REGION Network 6: Генерация импульса 10 сек.
   RUNG wire#powerrail
      { S7_Templates := "SrcType := Int" } NE_Contact(in1 := "Time_SYS_DB".Time_Now.Second, in2 := #last_10s)
      Mod(in1 := "Time_SYS_DB".Time_Now.Second, in2 := 10, out => #cnt_10s)
      wire#w1
      { S7_Templates := "SrcType := Int" } EQ_Contact(in1 := "Time_SYS_DB".Time_Now.Second, in2 := 0)
      wire#w2
      Move(in := "Time_SYS_DB".Time_Now.Second, out1 => #last_10s)
      Coil( "pulse_10s" )
   END_RUNG
   RUNG wire#w1
      { S7_Templates := "SrcType := Int" } EQ_Contact(in1 := #cnt_10s, in2 := 0)
   END_RUNG wire#w2
   // the same network as SCL:
   #_w1 := "Time_SYS_DB".Time_Now.Second <> #last_10s;
   IF #_w1 THEN #cnt_10s := "Time_SYS_DB".Time_Now.Second MOD 10; END_IF;
   #_w2 := #_w1 AND (("Time_SYS_DB".Time_Now.Second = 0) OR (#cnt_10s = 0));
   IF #_w2 THEN #last_10s := "Time_SYS_DB".Time_Now.Second; END_IF;
   "pulse_10s" := #_w2;
END_REGION

REGION Network 7: Генерация импульса 30 сек.
   RUNG wire#powerrail
      { S7_Templates := "SrcType := Int" } NE_Contact(in1 := "Time_SYS_DB".Time_Now.Second, in2 := #last_30s)
      Mod(in1 := "Time_SYS_DB".Time_Now.Second, in2 := 30, out => #cnt_30s)
      wire#w1
      { S7_Templates := "SrcType := Int" } EQ_Contact(in1 := "Time_SYS_DB".Time_Now.Second, in2 := 0)
      wire#w2
      Move(in := "Time_SYS_DB".Time_Now.Second, out1 => #last_30s)
      Coil( "pulse_30s" )
   END_RUNG
   RUNG wire#w1
      { S7_Templates := "SrcType := Int" } EQ_Contact(in1 := #cnt_30s, in2 := 0)
   END_RUNG wire#w2
   // the same network as SCL:
   #_w1 := "Time_SYS_DB".Time_Now.Second <> #last_30s;
   IF #_w1 THEN #cnt_30s := "Time_SYS_DB".Time_Now.Second MOD 30; END_IF;
   #_w2 := #_w1 AND (("Time_SYS_DB".Time_Now.Second = 0) OR (#cnt_30s = 0));
   IF #_w2 THEN #last_30s := "Time_SYS_DB".Time_Now.Second; END_IF;
   "pulse_30s" := #_w2;
END_REGION

REGION Network 8: Генерация импульса 1 мин.
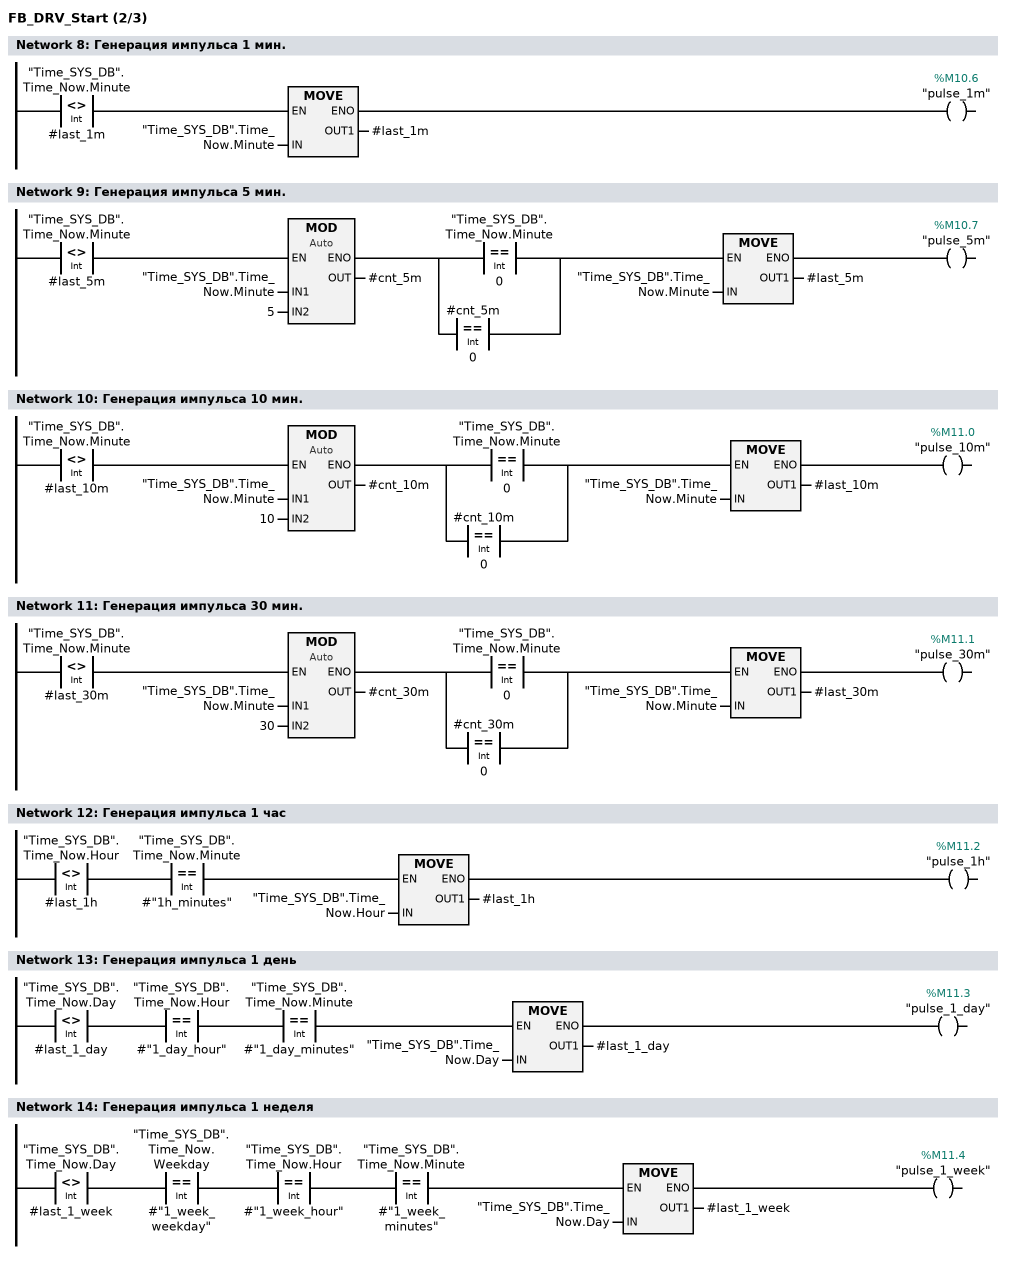
   RUNG wire#powerrail
      { S7_Templates := "SrcType := Int" } NE_Contact(in1 := "Time_SYS_DB".Time_Now.Minute, in2 := #last_1m)
      Move(in := "Time_SYS_DB".Time_Now.Minute, out1 => #last_1m)
      Coil( "pulse_1m" )
   END_RUNG
   // the same network as SCL:
   #_w1 := "Time_SYS_DB".Time_Now.Minute <> #last_1m;
   IF #_w1 THEN #last_1m := "Time_SYS_DB".Time_Now.Minute; END_IF;
   "pulse_1m" := #_w1;
END_REGION

REGION Network 9: Генерация импульса 5 мин.
   RUNG wire#powerrail
      { S7_Templates := "SrcType := Int" } NE_Contact(in1 := "Time_SYS_DB".Time_Now.Minute, in2 := #last_5m)
      Mod(in1 := "Time_SYS_DB".Time_Now.Minute, in2 := 5, out => #cnt_5m)
      wire#w1
      { S7_Templates := "SrcType := Int" } EQ_Contact(in1 := "Time_SYS_DB".Time_Now.Minute, in2 := 0)
      wire#w2
      Move(in := "Time_SYS_DB".Time_Now.Minute, out1 => #last_5m)
      Coil( "pulse_5m" )
   END_RUNG
   RUNG wire#w1
      { S7_Templates := "SrcType := Int" } EQ_Contact(in1 := #cnt_5m, in2 := 0)
   END_RUNG wire#w2
   // the same network as SCL:
   #_w1 := "Time_SYS_DB".Time_Now.Minute <> #last_5m;
   IF #_w1 THEN #cnt_5m := "Time_SYS_DB".Time_Now.Minute MOD 5; END_IF;
   #_w2 := #_w1 AND (("Time_SYS_DB".Time_Now.Minute = 0) OR (#cnt_5m = 0));
   IF #_w2 THEN #last_5m := "Time_SYS_DB".Time_Now.Minute; END_IF;
   "pulse_5m" := #_w2;
END_REGION

REGION Network 10: Генерация импульса 10 мин.
   RUNG wire#powerrail
      { S7_Templates := "SrcType := Int" } NE_Contact(in1 := "Time_SYS_DB".Time_Now.Minute, in2 := #last_10m)
      Mod(in1 := "Time_SYS_DB".Time_Now.Minute, in2 := 10, out => #cnt_10m)
      wire#w1
      { S7_Templates := "SrcType := Int" } EQ_Contact(in1 := "Time_SYS_DB".Time_Now.Minute, in2 := 0)
      wire#w2
      Move(in := "Time_SYS_DB".Time_Now.Minute, out1 => #last_10m)
      Coil( "pulse_10m" )
   END_RUNG
   RUNG wire#w1
      { S7_Templates := "SrcType := Int" } EQ_Contact(in1 := #cnt_10m, in2 := 0)
   END_RUNG wire#w2
   // the same network as SCL:
   #_w1 := "Time_SYS_DB".Time_Now.Minute <> #last_10m;
   IF #_w1 THEN #cnt_10m := "Time_SYS_DB".Time_Now.Minute MOD 10; END_IF;
   #_w2 := #_w1 AND (("Time_SYS_DB".Time_Now.Minute = 0) OR (#cnt_10m = 0));
   IF #_w2 THEN #last_10m := "Time_SYS_DB".Time_Now.Minute; END_IF;
   "pulse_10m" := #_w2;
END_REGION

REGION Network 11: Генерация импульса 30 мин.
   RUNG wire#powerrail
      { S7_Templates := "SrcType := Int" } NE_Contact(in1 := "Time_SYS_DB".Time_Now.Minute, in2 := #last_30m)
      Mod(in1 := "Time_SYS_DB".Time_Now.Minute, in2 := 30, out => #cnt_30m)
      wire#w1
      { S7_Templates := "SrcType := Int" } EQ_Contact(in1 := "Time_SYS_DB".Time_Now.Minute, in2 := 0)
      wire#w2
      Move(in := "Time_SYS_DB".Time_Now.Minute, out1 => #last_30m)
      Coil( "pulse_30m" )
   END_RUNG
   RUNG wire#w1
      { S7_Templates := "SrcType := Int" } EQ_Contact(in1 := #cnt_30m, in2 := 0)
   END_RUNG wire#w2
   // the same network as SCL:
   #_w1 := "Time_SYS_DB".Time_Now.Minute <> #last_30m;
   IF #_w1 THEN #cnt_30m := "Time_SYS_DB".Time_Now.Minute MOD 30; END_IF;
   #_w2 := #_w1 AND (("Time_SYS_DB".Time_Now.Minute = 0) OR (#cnt_30m = 0));
   IF #_w2 THEN #last_30m := "Time_SYS_DB".Time_Now.Minute; END_IF;
   "pulse_30m" := #_w2;
END_REGION

REGION Network 12: Генерация импульса 1 час
   RUNG wire#powerrail
      { S7_Templates := "SrcType := Int" } NE_Contact(in1 := "Time_SYS_DB".Time_Now.Hour, in2 := #last_1h)
      { S7_Templates := "SrcType := Int" } EQ_Contact(in1 := "Time_SYS_DB".Time_Now.Minute, in2 := #"1h_minutes")
      Move(in := "Time_SYS_DB".Time_Now.Hour, out1 => #last_1h)
      Coil( "pulse_1h" )
   END_RUNG
   // the same network as SCL:
   #_w1 := ("Time_SYS_DB".Time_Now.Hour <> #last_1h) AND ("Time_SYS_DB".Time_Now.Minute = #"1h_minutes");
   IF #_w1 THEN #last_1h := "Time_SYS_DB".Time_Now.Hour; END_IF;
   "pulse_1h" := #_w1;
END_REGION

REGION Network 13: Генерация импульса 1 день
   RUNG wire#powerrail
      { S7_Templates := "SrcType := Int" } NE_Contact(in1 := "Time_SYS_DB".Time_Now.Day, in2 := #last_1_day)
      { S7_Templates := "SrcType := Int" } EQ_Contact(in1 := "Time_SYS_DB".Time_Now.Hour, in2 := #"1_day_hour")
      { S7_Templates := "SrcType := Int" } EQ_Contact(in1 := "Time_SYS_DB".Time_Now.Minute, in2 := #"1_day_minutes")
      Move(in := "Time_SYS_DB".Time_Now.Day, out1 => #last_1_day)
      Coil( "pulse_1_day" )
   END_RUNG
   // the same network as SCL:
   #_w1 := ("Time_SYS_DB".Time_Now.Day <> #last_1_day) AND ("Time_SYS_DB".Time_Now.Hour = #"1_day_hour") AND ("Time_SYS_DB".Time_Now.Minute = #"1_day_minutes");
   IF #_w1 THEN #last_1_day := "Time_SYS_DB".Time_Now.Day; END_IF;
   "pulse_1_day" := #_w1;
END_REGION

REGION Network 14: Генерация импульса 1 неделя
   RUNG wire#powerrail
      { S7_Templates := "SrcType := Int" } NE_Contact(in1 := "Time_SYS_DB".Time_Now.Day, in2 := #last_1_week)
      { S7_Templates := "SrcType := Int" } EQ_Contact(in1 := "Time_SYS_DB".Time_Now.Weekday, in2 := #"1_week_weekday")
      { S7_Templates := "SrcType := Int" } EQ_Contact(in1 := "Time_SYS_DB".Time_Now.Hour, in2 := #"1_week_hour")
      { S7_Templates := "SrcType := Int" } EQ_Contact(in1 := "Time_SYS_DB".Time_Now.Minute, in2 := #"1_week_minutes")
      Move(in := "Time_SYS_DB".Time_Now.Day, out1 => #last_1_week)
      Coil( "pulse_1_week" )
   END_RUNG
   // the same network as SCL:
   #_w1 := ("Time_SYS_DB".Time_Now.Day <> #last_1_week) AND ("Time_SYS_DB".Time_Now.Weekday = #"1_week_weekday") AND ("Time_SYS_DB".Time_Now.Hour = #"1_week_hour") AND ("Time_SYS_DB".Time_Now.Minute = #"1_week_minutes");
   IF #_w1 THEN #last_1_week := "Time_SYS_DB".Time_Now.Day; END_IF;
   "pulse_1_week" := #_w1;
END_REGION

REGION Network 15: Генерация импульса 1 месяц
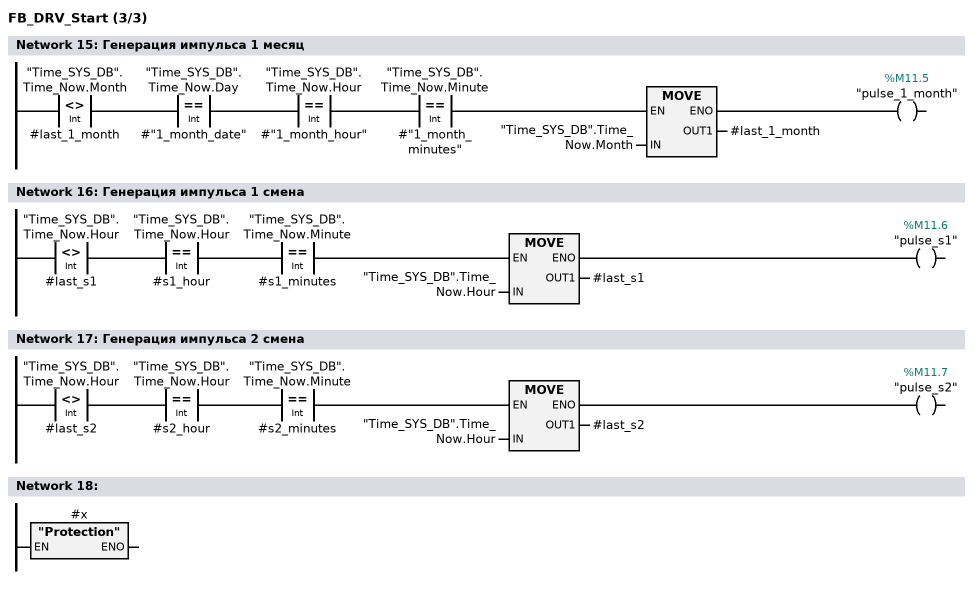
   RUNG wire#powerrail
      { S7_Templates := "SrcType := Int" } NE_Contact(in1 := "Time_SYS_DB".Time_Now.Month, in2 := #last_1_month)
      { S7_Templates := "SrcType := Int" } EQ_Contact(in1 := "Time_SYS_DB".Time_Now.Day, in2 := #"1_month_date")
      { S7_Templates := "SrcType := Int" } EQ_Contact(in1 := "Time_SYS_DB".Time_Now.Hour, in2 := #"1_month_hour")
      { S7_Templates := "SrcType := Int" } EQ_Contact(in1 := "Time_SYS_DB".Time_Now.Minute, in2 := #"1_month_minutes")
      Move(in := "Time_SYS_DB".Time_Now.Month, out1 => #last_1_month)
      Coil( "pulse_1_month" )
   END_RUNG
   // the same network as SCL:
   #_w1 := ("Time_SYS_DB".Time_Now.Month <> #last_1_month) AND ("Time_SYS_DB".Time_Now.Day = #"1_month_date") AND ("Time_SYS_DB".Time_Now.Hour = #"1_month_hour") AND ("Time_SYS_DB".Time_Now.Minute = #"1_month_minutes");
   IF #_w1 THEN #last_1_month := "Time_SYS_DB".Time_Now.Month; END_IF;
   "pulse_1_month" := #_w1;
END_REGION

REGION Network 16: Генерация импульса 1 смена
   RUNG wire#powerrail
      { S7_Templates := "SrcType := Int" } NE_Contact(in1 := "Time_SYS_DB".Time_Now.Hour, in2 := #last_s1)
      { S7_Templates := "SrcType := Int" } EQ_Contact(in1 := "Time_SYS_DB".Time_Now.Hour, in2 := #s1_hour)
      { S7_Templates := "SrcType := Int" } EQ_Contact(in1 := "Time_SYS_DB".Time_Now.Minute, in2 := #s1_minutes)
      Move(in := "Time_SYS_DB".Time_Now.Hour, out1 => #last_s1)
      Coil( "pulse_s1" )
   END_RUNG
   // the same network as SCL:
   #_w1 := ("Time_SYS_DB".Time_Now.Hour <> #last_s1) AND ("Time_SYS_DB".Time_Now.Hour = #s1_hour) AND ("Time_SYS_DB".Time_Now.Minute = #s1_minutes);
   IF #_w1 THEN #last_s1 := "Time_SYS_DB".Time_Now.Hour; END_IF;
   "pulse_s1" := #_w1;
END_REGION

REGION Network 17: Генерация импульса 2 смена
   RUNG wire#powerrail
      { S7_Templates := "SrcType := Int" } NE_Contact(in1 := "Time_SYS_DB".Time_Now.Hour, in2 := #last_s2)
      { S7_Templates := "SrcType := Int" } EQ_Contact(in1 := "Time_SYS_DB".Time_Now.Hour, in2 := #s2_hour)
      { S7_Templates := "SrcType := Int" } EQ_Contact(in1 := "Time_SYS_DB".Time_Now.Minute, in2 := #s2_minutes)
      Move(in := "Time_SYS_DB".Time_Now.Hour, out1 => #last_s2)
      Coil( "pulse_s2" )
   END_RUNG
   // the same network as SCL:
   #_w1 := ("Time_SYS_DB".Time_Now.Hour <> #last_s2) AND ("Time_SYS_DB".Time_Now.Hour = #s2_hour) AND ("Time_SYS_DB".Time_Now.Minute = #s2_minutes);
   IF #_w1 THEN #last_s2 := "Time_SYS_DB".Time_Now.Hour; END_IF;
   "pulse_s2" := #_w1;
END_REGION

REGION Network 18
   RUNG wire#powerrail
      #x()
   END_RUNG
   // the same network as SCL:
   #x();   // "Protection"
END_REGION
END_FUNCTION_BLOCK

FUNCTION_BLOCK "Time_SYS"   // FB95, LAD
{ S7_Optimized_Access := 'FALSE' }
VERSION : 0.1
// stored: AutoNumber false, IsIECCheckEnabled false, SetENOAutomatically false, UDAEnableTagReadback false
   VAR DB_SPECIFIC
      Set_Time : Bool;   // Заданное время
      Time_Now : Struct   // Текущее время
         Year : Int;   // год
         Month : Int;   // месяц
         Day : Int;   // день месяца
         Weekday : Int;   // день недели (1 - воскресенье)
         Hour : Int;   // часы
         Minute : Int;   // минуты
         Second : Int;   // секунды
      END_STRUCT;
      Time_SP : Struct   // Текущее время
         Year : Int;   // год
         Month : Int;   // месяц
         Day : Int;   // день месяца
         Weekday : Int;   // день недели (1 - воскресенье)
         Hour : Int;   // часы
         Minute : Int;   // минуты
         Second : Int;   // секунды
      END_STRUCT;
      TimeZone { S7_SetPoint := 'True'} : TimeTransformationRule;   // Часовой пояс
      RD_SYS_Status : Int;   // Статус чтения времени
      WR_SYS_Status : Int;   // Статус записи времени
      RD_Time : DTL;   // Прочитанное сист. время
      SP_Time : DTL;   // Новое сист. время
   END_VAR
   VAR
      SET_TIMEZONE { S7_SetPoint := 'True'} : SET_TIMEZONE;   // Запись часового пояса
   END_VAR
   VAR DB_SPECIFIC
      Time_DTL : DTL;
   END_VAR
   // TimeZone.Bias := 180;   // Часовой пояс по GMT (смещение в минутах)
   // TimeZone.DaylightBias := 60;
   // TimeZone.DaylightStartMonth := 3;
   // TimeZone.DaylightStartWeek := 5;
   // TimeZone.DaylightStartWeekday := 7;
   // TimeZone.DaylightStartHour := 2;
   // TimeZone.DaylightStartMinute := 0;
   // TimeZone.StandardStartMonth := 10;
   // TimeZone.StandardStartWeek := 5;
   // TimeZone.StandardStartWeekday := 1;
   // TimeZone.StandardStartHour := 3;
   // TimeZone.StandardStartMinute := 0;
   // TimeZone.TimeZoneName := 'GMT+3';
   VAR_TEMP   // added for the SCL form of the ladder/FBD networks
      _w1 : Bool;
   END_VAR
BEGIN

REGION Network 1: Чтение системного времени
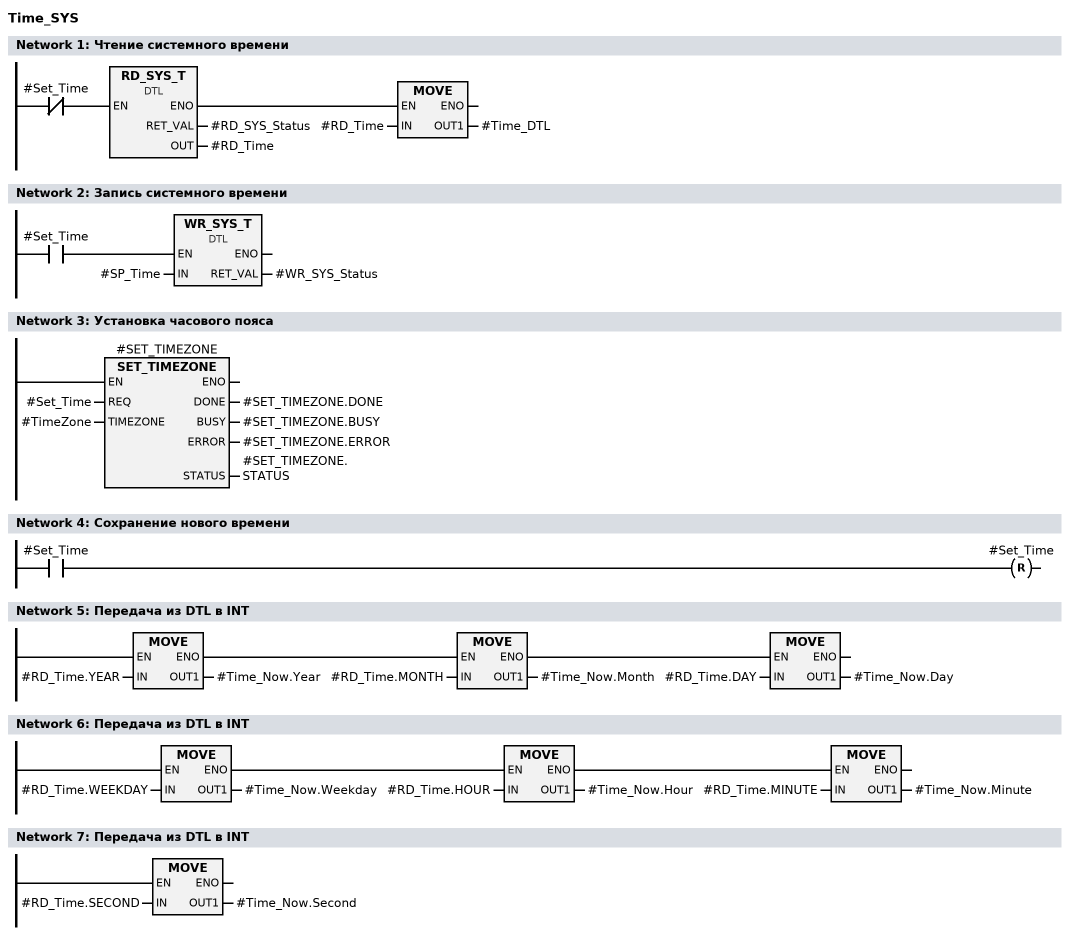
   RUNG wire#powerrail
      I_Contact( #Set_Time )
      { S7_Templates := "date_type := DTL" } RD_SYS_T(RET_VAL => #RD_SYS_Status, OUT => #RD_Time)
      Move(in := #RD_Time, out1 => #Time_DTL)
   END_RUNG
   // the same network as SCL:
   #RD_SYS_Status := RD_SYS_T(EN := NOT #Set_Time, OUT => #RD_Time, ENO => #_w1);
   IF #_w1 THEN #Time_DTL := #RD_Time; END_IF;
END_REGION

REGION Network 2: Запись системного времени
   RUNG wire#powerrail
      Contact( #Set_Time )
      { S7_Templates := "date_type := DTL" } WR_SYS_T(IN := #SP_Time, RET_VAL => #WR_SYS_Status)
   END_RUNG
   // the same network as SCL:
   IF #Set_Time THEN #WR_SYS_Status := WR_SYS_T(IN := #SP_Time); END_IF;
END_REGION

REGION Network 3: Установка часового пояса
   RUNG wire#powerrail
      #SET_TIMEZONE.SET_TIMEZONE(REQ := #Set_Time, TimeZone := #TimeZone, DONE => #SET_TIMEZONE.DONE, BUSY => #SET_TIMEZONE.BUSY, ERROR => #SET_TIMEZONE.ERROR, STATUS => #SET_TIMEZONE.STATUS)
   END_RUNG
   // the same network as SCL:
   #SET_TIMEZONE(REQ := #Set_Time,   // SET_TIMEZONE
                 TimeZone := #TimeZone,
                 DONE => #SET_TIMEZONE.DONE,
                 BUSY => #SET_TIMEZONE.BUSY,
                 ERROR => #SET_TIMEZONE.ERROR,
                 STATUS => #SET_TIMEZONE.STATUS);
END_REGION

REGION Network 4: Сохранение нового времени
   RUNG wire#powerrail
      Contact( #Set_Time )
      R_Coil( #Set_Time )
   END_RUNG
   // the same network as SCL:
   IF #Set_Time THEN #Set_Time := FALSE; END_IF;
END_REGION

REGION Network 5: Передача из DTL в INT
   RUNG wire#powerrail
      Move(in := #RD_Time.YEAR, out1 => #Time_Now.Year)
      Move(in := #RD_Time.MONTH, out1 => #Time_Now.Month)
      Move(in := #RD_Time.DAY, out1 => #Time_Now.Day)
   END_RUNG
   // the same network as SCL:
   #Time_Now.Year := #RD_Time.YEAR;
   #Time_Now.Month := #RD_Time.MONTH;
   #Time_Now.Day := #RD_Time.DAY;
END_REGION

REGION Network 6: Передача из DTL в INT
   RUNG wire#powerrail
      Move(in := #RD_Time.WEEKDAY, out1 => #Time_Now.Weekday)
      Move(in := #RD_Time.HOUR, out1 => #Time_Now.Hour)
      Move(in := #RD_Time.MINUTE, out1 => #Time_Now.Minute)
   END_RUNG
   // the same network as SCL:
   #Time_Now.Weekday := #RD_Time.WEEKDAY;
   #Time_Now.Hour := #RD_Time.HOUR;
   #Time_Now.Minute := #RD_Time.MINUTE;
END_REGION

REGION Network 7: Передача из DTL в INT
   RUNG wire#powerrail
      Move(in := #RD_Time.SECOND, out1 => #Time_Now.Second)
   END_RUNG
   // the same network as SCL:
   #Time_Now.Second := #RD_Time.SECOND;
END_REGION
END_FUNCTION_BLOCK

FUNCTION_BLOCK "Time_D"   // FB94, LAD
{ S7_Optimized_Access := 'FALSE' }
VERSION : 0.1
// stored: AutoNumber false, IsIECCheckEnabled false, SetENOAutomatically false, UDAEnableTagReadback false
   VAR DB_SPECIFIC
      SP_D { S7_SetPoint := 'True'} : DInt := 4;   // Уставка дней - от 0 до 999
      SP_H { S7_SetPoint := 'True'} : DInt;   // Уставка часов - от 0 до 23
      SP_M { S7_SetPoint := 'True'} : DInt;   // Уставка минут - от 0 до 59
      SP_S { S7_SetPoint := 'True'} : DInt;   // Уставка секунд - от 0 до 59
      Now_D : DInt;   // Прошло дней от начала отсчёта
      Now_H : DInt;   // Прошло часов от начала отсчёта
      Now_M : DInt;   // Прошло минут от начала отсчёта
      Now_S : DInt;   // Прошло секунд от начала отсчёта
      Rev_D : DInt;   // Осталось дней до уставки
      Rev_H : DInt;   // Осталось часов до уставки
      Rev_M : DInt;   // Осталось минут до уставки
      Rev_S : DInt;   // Осталось секунд до уставки
      Progress : Real;   // Прогресс выполнения
      Start : Bool;   // Запуск
      "Exit" : Bool;   // Счёт завершён
      Pause : Bool;   // Пауза
      Reset : Bool;   // Сброс таймера
   END_VAR
   VAR_TEMP
      Full_SP_S : DInt;
      Full_Now_S : DInt;
      Full_Delta_S : DInt;
      x1 : DInt;
      x2 : DInt;
   END_VAR
   VAR_TEMP   // added for the SCL form of the ladder/FBD networks
      _w1 : Bool;
      _w2 : Bool;
      _w3 : Bool;
   END_VAR
BEGIN

REGION Network 1: Подсчёт времени
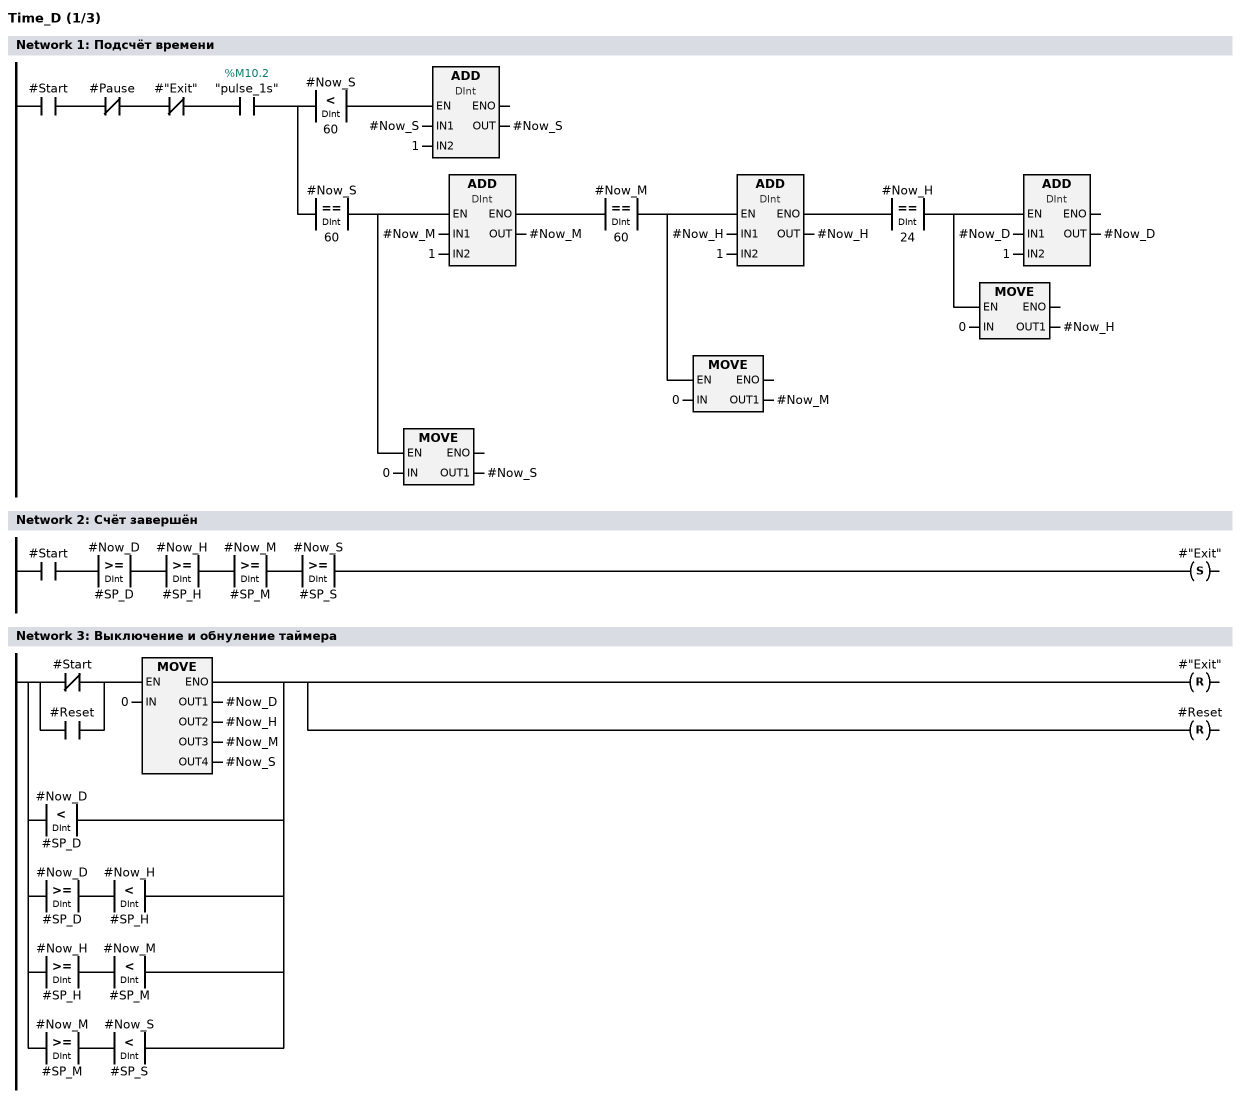
   RUNG wire#powerrail
      Contact( #Start )
      I_Contact( #Pause )
      I_Contact( #"Exit" )
      Contact( "pulse_1s" )
      wire#w1
      { S7_Templates := "SrcType := DInt" } LT_Contact(in1 := #Now_S, in2 := 60)
      { S7_Templates := "SrcType := DInt"; S7_GenerateENO := "TRUE" } Add(in1 := #Now_S, in2 := 1, out => #Now_S)
   END_RUNG
   RUNG wire#w1
      { S7_Templates := "SrcType := DInt" } EQ_Contact(in1 := #Now_S, in2 := 60)
      wire#w2
      { S7_Templates := "SrcType := DInt"; S7_GenerateENO := "TRUE" } Add(in1 := #Now_M, in2 := 1, out => #Now_M)
      { S7_Templates := "SrcType := DInt" } EQ_Contact(in1 := #Now_M, in2 := 60)
      wire#w3
      { S7_Templates := "SrcType := DInt"; S7_GenerateENO := "TRUE" } Add(in1 := #Now_H, in2 := 1, out => #Now_H)
      { S7_Templates := "SrcType := DInt" } EQ_Contact(in1 := #Now_H, in2 := 24)
      wire#w4
      { S7_Templates := "SrcType := DInt"; S7_GenerateENO := "TRUE" } Add(in1 := #Now_D, in2 := 1, out => #Now_D)
   END_RUNG
   RUNG wire#w4
      { S7_GenerateENO := "TRUE" } Move(in := 0, out1 => #Now_H)
   END_RUNG
   RUNG wire#w3
      { S7_GenerateENO := "TRUE" } Move(in := 0, out1 => #Now_M)
   END_RUNG
   RUNG wire#w2
      { S7_GenerateENO := "TRUE" } Move(in := 0, out1 => #Now_S)
   END_RUNG
   // the same network as SCL:
   // ENO of a box is taken as its EN; it also drops when the box reports an error
   #_w1 := #Start AND NOT #Pause AND NOT #"Exit" AND "pulse_1s";
   IF #_w1 AND (#Now_S < 60) THEN #Now_S := #Now_S + 1; END_IF;
   #_w2 := #_w1 AND (#Now_S = 60);
   IF #_w2 THEN #Now_M := #Now_M + 1; END_IF;
   #_w3 := #_w2 AND (#Now_M = 60);
   IF #_w3 THEN #Now_H := #Now_H + 1; END_IF;
   IF #_w3 AND (#Now_H = 24) THEN
       #Now_D := #Now_D + 1;
       #Now_H := 0;
   END_IF;
   IF #_w3 THEN #Now_M := 0; END_IF;
   IF #_w2 THEN #Now_S := 0; END_IF;
END_REGION

REGION Network 2: Счёт завершён
   RUNG wire#powerrail
      Contact( #Start )
      { S7_Templates := "SrcType := DInt" } GE_Contact(in1 := #Now_D, in2 := #SP_D)
      { S7_Templates := "SrcType := DInt" } GE_Contact(in1 := #Now_H, in2 := #SP_H)
      { S7_Templates := "SrcType := DInt" } GE_Contact(in1 := #Now_M, in2 := #SP_M)
      { S7_Templates := "SrcType := DInt" } GE_Contact(in1 := #Now_S, in2 := #SP_S)
      S_Coil( #"Exit" )
   END_RUNG
   // the same network as SCL:
   IF #Start AND (#Now_D >= #SP_D) AND (#Now_H >= #SP_H) AND (#Now_M >= #SP_M) AND (#Now_S >= #SP_S) THEN
       #"Exit" := TRUE;
   END_IF;
END_REGION

REGION Network 3: Выключение и обнуление таймера
   RUNG wire#powerrail
      I_Contact( #Start )
      wire#w1
      { S7_GenerateENO := "TRUE" } Move(in := 0, out1 => #Now_D, out2 => #Now_H, out3 => #Now_M, out4 => #Now_S)
      wire#w2
      R_Coil( #"Exit" )
   END_RUNG
   RUNG wire#powerrail
      Contact( #Reset )
   END_RUNG wire#w1
   RUNG wire#powerrail
      { S7_Templates := "SrcType := DInt" } LT_Contact(in1 := #Now_D, in2 := #SP_D)
   END_RUNG wire#w2
   RUNG wire#powerrail
      { S7_Templates := "SrcType := DInt" } GE_Contact(in1 := #Now_D, in2 := #SP_D)
      { S7_Templates := "SrcType := DInt" } LT_Contact(in1 := #Now_H, in2 := #SP_H)
   END_RUNG wire#w2
   RUNG wire#powerrail
      { S7_Templates := "SrcType := DInt" } GE_Contact(in1 := #Now_H, in2 := #SP_H)
      { S7_Templates := "SrcType := DInt" } LT_Contact(in1 := #Now_M, in2 := #SP_M)
   END_RUNG wire#w2
   RUNG wire#powerrail
      { S7_Templates := "SrcType := DInt" } GE_Contact(in1 := #Now_M, in2 := #SP_M)
      { S7_Templates := "SrcType := DInt" } LT_Contact(in1 := #Now_S, in2 := #SP_S)
   END_RUNG wire#w2
   RUNG wire#w2
      R_Coil( #Reset )
   END_RUNG
   // the same network as SCL:
   // ENO of a box is taken as its EN; it also drops when the box reports an error
   #_w1 := NOT #Start OR #Reset;
   IF #_w1 THEN
       #Now_D := 0;
       #Now_H := 0;
       #Now_M := 0;
       #Now_S := 0;
   END_IF;
   IF #_w1 OR (#Now_D < #SP_D) OR ((#Now_D >= #SP_D) AND (#Now_H < #SP_H)) OR ((#Now_H >= #SP_H) AND (#Now_M < #SP_M)) OR ((#Now_M >= #SP_M) AND (#Now_S < #SP_S)) THEN
       #"Exit" := FALSE;
       #Reset := FALSE;
   END_IF;
END_REGION

REGION Network 4: Поправка переполнения времени
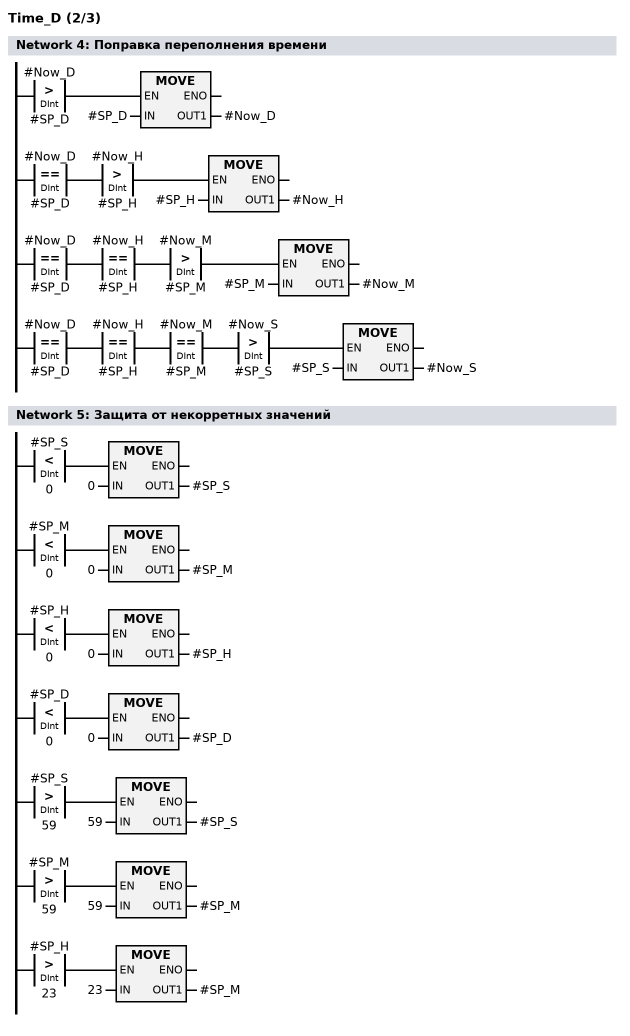
   RUNG wire#powerrail
      { S7_Templates := "SrcType := DInt" } GT_Contact(in1 := #Now_D, in2 := #SP_D)
      { S7_GenerateENO := "TRUE" } Move(in := #SP_D, out1 => #Now_D)
   END_RUNG
   RUNG wire#powerrail
      { S7_Templates := "SrcType := DInt" } EQ_Contact(in1 := #Now_D, in2 := #SP_D)
      { S7_Templates := "SrcType := DInt" } GT_Contact(in1 := #Now_H, in2 := #SP_H)
      { S7_GenerateENO := "TRUE" } Move(in := #SP_H, out1 => #Now_H)
   END_RUNG
   RUNG wire#powerrail
      { S7_Templates := "SrcType := DInt" } EQ_Contact(in1 := #Now_D, in2 := #SP_D)
      { S7_Templates := "SrcType := DInt" } EQ_Contact(in1 := #Now_H, in2 := #SP_H)
      { S7_Templates := "SrcType := DInt" } GT_Contact(in1 := #Now_M, in2 := #SP_M)
      { S7_GenerateENO := "TRUE" } Move(in := #SP_M, out1 => #Now_M)
   END_RUNG
   RUNG wire#powerrail
      { S7_Templates := "SrcType := DInt" } EQ_Contact(in1 := #Now_D, in2 := #SP_D)
      { S7_Templates := "SrcType := DInt" } EQ_Contact(in1 := #Now_H, in2 := #SP_H)
      { S7_Templates := "SrcType := DInt" } EQ_Contact(in1 := #Now_M, in2 := #SP_M)
      { S7_Templates := "SrcType := DInt" } GT_Contact(in1 := #Now_S, in2 := #SP_S)
      { S7_GenerateENO := "TRUE" } Move(in := #SP_S, out1 => #Now_S)
   END_RUNG
   // the same network as SCL:
   IF #Now_D > #SP_D THEN #Now_D := #SP_D; END_IF;
   IF (#Now_D = #SP_D) AND (#Now_H > #SP_H) THEN #Now_H := #SP_H; END_IF;
   IF (#Now_D = #SP_D) AND (#Now_H = #SP_H) AND (#Now_M > #SP_M) THEN #Now_M := #SP_M; END_IF;
   IF (#Now_D = #SP_D) AND (#Now_H = #SP_H) AND (#Now_M = #SP_M) AND (#Now_S > #SP_S) THEN
       #Now_S := #SP_S;
   END_IF;
END_REGION

REGION Network 5: Защита от некорретных значений
   RUNG wire#powerrail
      { S7_Templates := "SrcType := DInt" } LT_Contact(in1 := #SP_S, in2 := 0)
      { S7_GenerateENO := "TRUE" } Move(in := 0, out1 => #SP_S)
   END_RUNG
   RUNG wire#powerrail
      { S7_Templates := "SrcType := DInt" } LT_Contact(in1 := #SP_M, in2 := 0)
      { S7_GenerateENO := "TRUE" } Move(in := 0, out1 => #SP_M)
   END_RUNG
   RUNG wire#powerrail
      { S7_Templates := "SrcType := DInt" } LT_Contact(in1 := #SP_H, in2 := 0)
      { S7_GenerateENO := "TRUE" } Move(in := 0, out1 => #SP_H)
   END_RUNG
   RUNG wire#powerrail
      { S7_Templates := "SrcType := DInt" } LT_Contact(in1 := #SP_D, in2 := 0)
      { S7_GenerateENO := "TRUE" } Move(in := 0, out1 => #SP_D)
   END_RUNG
   RUNG wire#powerrail
      { S7_Templates := "SrcType := DInt" } GT_Contact(in1 := #SP_S, in2 := 59)
      { S7_GenerateENO := "TRUE" } Move(in := 59, out1 => #SP_S)
   END_RUNG
   RUNG wire#powerrail
      { S7_Templates := "SrcType := DInt" } GT_Contact(in1 := #SP_M, in2 := 59)
      { S7_GenerateENO := "TRUE" } Move(in := 59, out1 => #SP_M)
   END_RUNG
   RUNG wire#powerrail
      { S7_Templates := "SrcType := DInt" } GT_Contact(in1 := #SP_H, in2 := 23)
      { S7_GenerateENO := "TRUE" } Move(in := 23, out1 => #SP_M)
   END_RUNG
   // the same network as SCL:
   IF #SP_S < 0 THEN #SP_S := 0; END_IF;
   IF #SP_M < 0 THEN #SP_M := 0; END_IF;
   IF #SP_H < 0 THEN #SP_H := 0; END_IF;
   IF #SP_D < 0 THEN #SP_D := 0; END_IF;
   IF #SP_S > 59 THEN #SP_S := 59; END_IF;
   IF #SP_M > 59 THEN #SP_M := 59; END_IF;
   IF #SP_H > 23 THEN #SP_M := 23; END_IF;
END_REGION

REGION Network 6: Обратный отсчёт
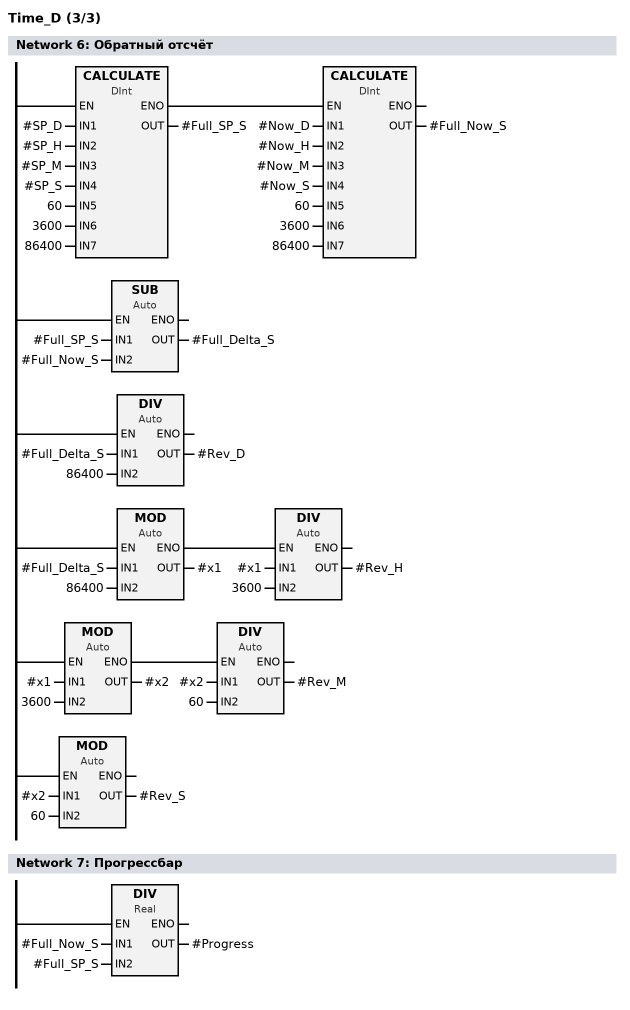
   RUNG wire#powerrail
      { S7_Templates := "SrcType := DInt"; S7_Expression := "(IN1*IN7)+(IN2*IN6)+(IN3*IN5)+IN4" } Calculate(in1 := #SP_D, in2 := #SP_H, in3 := #SP_M, in4 := #SP_S, in5 := 60, in6 := 3600, in7 := 86400, out => #Full_SP_S)
      { S7_Templates := "SrcType := DInt"; S7_Expression := "(IN1*IN7)+(IN2*IN6)+(IN3*IN5)+IN4" } Calculate(in1 := #Now_D, in2 := #Now_H, in3 := #Now_M, in4 := #Now_S, in5 := 60, in6 := 3600, in7 := 86400, out => #Full_Now_S)
   END_RUNG
   RUNG wire#powerrail
      Sub(in1 := #Full_SP_S, in2 := #Full_Now_S, out => #Full_Delta_S)
   END_RUNG
   RUNG wire#powerrail
      Div(in1 := #Full_Delta_S, in2 := 86400, out => #Rev_D)
   END_RUNG
   RUNG wire#powerrail
      Mod(in1 := #Full_Delta_S, in2 := 86400, out => #x1)
      Div(in1 := #x1, in2 := 3600, out => #Rev_H)
   END_RUNG
   RUNG wire#powerrail
      Mod(in1 := #x1, in2 := 3600, out => #x2)
      Div(in1 := #x2, in2 := 60, out => #Rev_M)
   END_RUNG
   RUNG wire#powerrail
      Mod(in1 := #x2, in2 := 60, out => #Rev_S)
   END_RUNG
   // the same network as SCL:
   #Full_SP_S := (#SP_D*86400)+(#SP_H*3600)+(#SP_M*60)+#SP_S;
   #Full_Now_S := (#Now_D*86400)+(#Now_H*3600)+(#Now_M*60)+#Now_S;
   #Full_Delta_S := #Full_SP_S - #Full_Now_S;
   #Rev_D := #Full_Delta_S / 86400;
   #x1 := #Full_Delta_S MOD 86400;
   #Rev_H := #x1 / 3600;
   #x2 := #x1 MOD 3600;
   #Rev_M := #x2 / 60;
   #Rev_S := #x2 MOD 60;
END_REGION

REGION Network 7: Прогрессбар
   RUNG wire#powerrail
      { S7_Templates := "SrcType := Real" } Div(in1 := #Full_Now_S, in2 := #Full_SP_S, out => #Progress)
   END_RUNG
   // the same network as SCL:
   #Progress := #Full_Now_S / #Full_SP_S;
END_REGION
END_FUNCTION_BLOCK

FUNCTION_BLOCK "DIx_1"   // FB200, LAD
{ S7_Optimized_Access := 'FALSE' }
VERSION : 0.1
// Input - входной сигнал контроллера
// pulse - частота фильтрации дребезга
// Signal - обработанный и отфильтрованный сигнал, используемый в дальнейшем
// stored: AutoNumber false, IsIECCheckEnabled false, SetENOAutomatically false, UDAEnableTagReadback false
   VAR
      AllBlock { S7_SetPoint := 'True'} : "DI_ex";   // Аварийный останов / 2.4 разрешение на работу
      EZ_1_FB_AHLS { S7_SetPoint := 'True'} : "DI_ex";   // Электролизер 1 (Переполнение поддона) / 2.3 Нижний уровень
      Gas_Chanel_1_1 { S7_SetPoint := 'True'} : "DI_ex";   // Загазованность канал 1 (Порог 1) / Ротаметр 1
      Gas_Chanel_1_2 { S7_SetPoint := 'True'} : "DI_ex";   // Загазованность канал 1 (Порог 2) / Ротаметр 2
      Gas_Chanel_2_1 { S7_SetPoint := 'True'} : "DI_ex";   // Загазованность канал 2 (Порог 1) / Ротаметр 3
      Gas_Chanel_2_2 { S7_SetPoint := 'True'} : "DI_ex";   // Загазованность канал 2 (Порог 2) / Датчик переливва
      ALS_1 { S7_SetPoint := 'True'} : "DI_ex";   // Аварийный уровень 1 / Датчик переливва
      KC_1 { S7_SetPoint := 'True'} : "DI_ex";   // Блок клапанов (Сигнал 1)
      KC_2 { S7_SetPoint := 'True'} : "DI_ex";   // Блок клапанов (Сигнал 2)
      signal_10 { S7_SetPoint := 'True'} : "DI_ex";
      signal_11 { S7_SetPoint := 'True'} : "DI_ex";
      signal_12 { S7_SetPoint := 'True'} : "DI_ex";
      signal_13 { S7_SetPoint := 'True'} : "DI_ex";
   END_VAR
   VAR DB_SPECIFIC
      Time_DTL { S7_SetPoint := 'True'} : DTL;
   END_VAR
   // AllBlock.ADDR_Byte := 1;
   // AllBlock.ADDR_Bit := 5;
   // EZ_1_FB_AHLS.ADDR_Byte := 0;
   // EZ_1_FB_AHLS.ADDR_Bit := 2;
   // Gas_Chanel_1_1.ADDR_Bit := 7;
   // Gas_Chanel_1_2.ADDR_Byte := 1;
   // Gas_Chanel_1_2.ADDR_Bit := 0;
   // Gas_Chanel_2_1.ADDR_Byte := 1;
   // Gas_Chanel_2_1.ADDR_Bit := 1;
   // Gas_Chanel_2_2.ADDR_Byte := 1;
   // Gas_Chanel_2_2.ADDR_Bit := 2;
   // ALS_1.ADDR_Byte := 2;
   // ALS_1.ADDR_Bit := 0;
   // KC_1.ADDR_Byte := 1;
   // KC_1.ADDR_Bit := 3;
   // KC_2.ADDR_Byte := 1;
   // KC_2.ADDR_Bit := 4;
   VAR_TEMP   // added for the SCL form of the ladder/FBD networks
      _w1 : Bool;
      _w2 : Bool;
   END_VAR
BEGIN

REGION Network 1: AllBlock
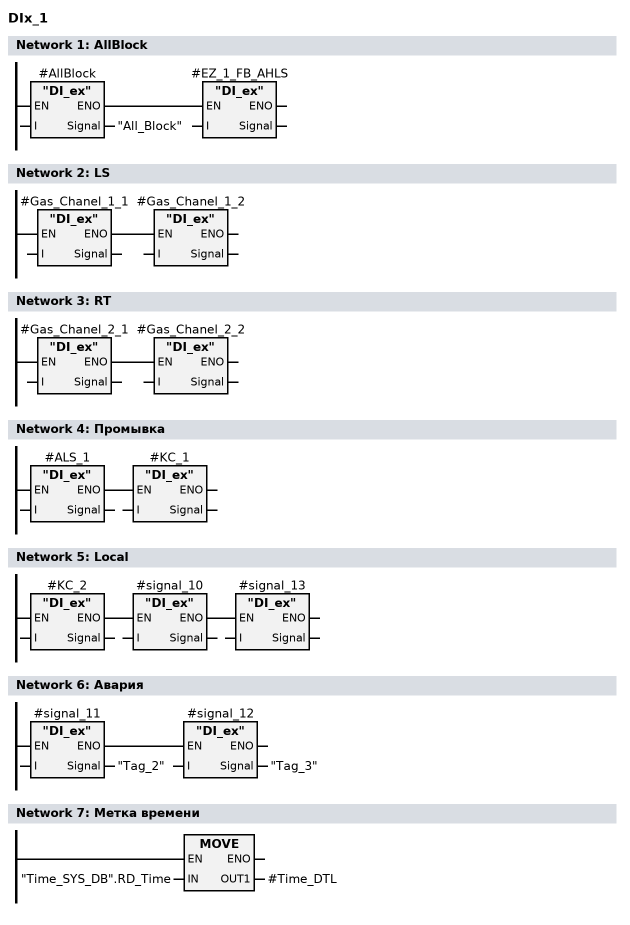
   RUNG wire#powerrail
      #AllBlock(I :=, Signal => "All_Block")
      #EZ_1_FB_AHLS(I :=, Signal =>)
   END_RUNG
   // the same network as SCL:
   #AllBlock(Signal => "All_Block", ENO => #_w1);   // "DI_ex"
   IF #_w1 THEN
       #EZ_1_FB_AHLS();   // "DI_ex"
   END_IF;
END_REGION

REGION Network 2: LS
   RUNG wire#powerrail
      #Gas_Chanel_1_1(I :=, Signal =>)
      #Gas_Chanel_1_2(I :=, Signal =>)
   END_RUNG
   // the same network as SCL:
   #Gas_Chanel_1_1(ENO => #_w1);   // "DI_ex"
   IF #_w1 THEN
       #Gas_Chanel_1_2();   // "DI_ex"
   END_IF;
END_REGION

REGION Network 3: RT
   RUNG wire#powerrail
      #Gas_Chanel_2_1(I :=, Signal =>)
      #Gas_Chanel_2_2(I :=, Signal =>)
   END_RUNG
   // the same network as SCL:
   #Gas_Chanel_2_1(ENO => #_w1);   // "DI_ex"
   IF #_w1 THEN
       #Gas_Chanel_2_2();   // "DI_ex"
   END_IF;
END_REGION

REGION Network 4: Промывка
   RUNG wire#powerrail
      #ALS_1(I :=, Signal =>)
      #KC_1(I :=, Signal =>)
   END_RUNG
   // the same network as SCL:
   #ALS_1(ENO => #_w1);   // "DI_ex"
   IF #_w1 THEN
       #KC_1();   // "DI_ex"
   END_IF;
END_REGION

REGION Network 5: Local
   RUNG wire#powerrail
      #KC_2(I :=, Signal =>)
      #signal_10(I :=, Signal =>)
      #signal_13(I :=, Signal =>)
   END_RUNG
   // the same network as SCL:
   #KC_2(ENO => #_w1);   // "DI_ex"
   #signal_10(EN := #_w1, ENO => #_w2);   // "DI_ex"
   IF #_w2 THEN
       #signal_13();   // "DI_ex"
   END_IF;
END_REGION

REGION Network 6: Авария
   RUNG wire#powerrail
      #signal_11(I :=, Signal => "Tag_2")
      #signal_12(I :=, Signal => "Tag_3")
   END_RUNG
   // the same network as SCL:
   #signal_11(Signal => "Tag_2", ENO => #_w1);   // "DI_ex"
   IF #_w1 THEN
       #signal_12(Signal => "Tag_3");   // "DI_ex"
   END_IF;
END_REGION

REGION Network 7: Метка времени
   RUNG wire#powerrail
      Move(in := "Time_SYS_DB".RD_Time, out1 => #Time_DTL)
   END_RUNG
   // the same network as SCL:
   #Time_DTL := "Time_SYS_DB".RD_Time;
END_REGION
END_FUNCTION_BLOCK

FUNCTION_BLOCK "DI_ex"   // FB101, LAD
{ S7_Optimized_Access := 'FALSE' }
VERSION : 0.1
// stored: AutoNumber false, IsIECCheckEnabled false, SetENOAutomatically false, UDAEnableTagReadback false
   VAR_INPUT
      I : Bool;   // Входной сигнал ПЛК
   END_VAR
   VAR_OUTPUT
      Signal : Bool;   // Результат обработки
   END_VAR
   VAR DB_SPECIFIC
      CMD : "CMD";   // Основные команды / Блок команд
      Use : Struct
         Inverse { S7_SetPoint := 'True'} : Bool;   // Инверсия входного сигнала
         Indirect { S7_SetPoint := 'True'} : Bool := true;   // Использование косвенной адресации
      END_STRUCT;
      ADDR_Byte { S7_SetPoint := 'True'} : Int;   // Адрес входа на контроллере (Байт)
      ADDR_Bit { S7_SetPoint := 'True'} : Int := 9;   // Адрес входа на контроллере (Бит)
   END_VAR
   VAR
      Filter_On { S7_SetPoint := 'True'} : "Time_S_b";   // Фильтр наличия сигнала
      Filter_Off { S7_SetPoint := 'True'} : "Time_S_b";   // Фильтр отсутствия сигнала
   END_VAR
   VAR_TEMP
      Data : Bool;
   END_VAR
   VAR_TEMP   // added for the SCL form of the ladder/FBD networks
      _w1 : Bool;
      _w2 : Bool;
   END_VAR
BEGIN

REGION Network 1: Устройство в ручном режиме
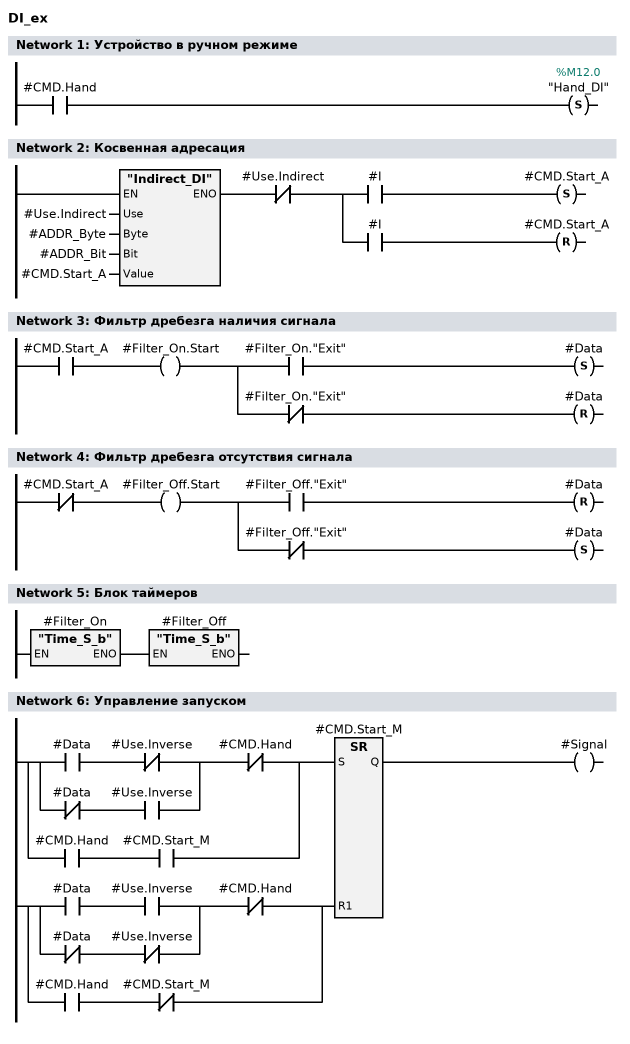
   RUNG wire#powerrail
      Contact( #CMD.Hand )
      S_Coil( "Hand_DI" )
   END_RUNG
   // the same network as SCL:
   IF #CMD.Hand THEN "Hand_DI" := TRUE; END_IF;
END_REGION

REGION Network 2: Косвенная адресация
   RUNG wire#powerrail
      "Indirect_DI"(Use := #Use.Indirect, "Byte" := #ADDR_Byte, Bit := #ADDR_Bit, Value := #CMD.Start_A)
      I_Contact( #Use.Indirect )
      wire#w1
      Contact( #I )
      S_Coil( #CMD.Start_A )
   END_RUNG
   RUNG wire#w1
      Contact( #I )
      R_Coil( #CMD.Start_A )
   END_RUNG
   // the same network as SCL:
   "Indirect_DI"(Use := #Use.Indirect,
                 "Byte" := #ADDR_Byte,
                 Bit := #ADDR_Bit,
                 Value := #CMD.Start_A,
                 ENO => #_w1);
   #_w2 := #_w1 AND NOT #Use.Indirect;
   IF #_w2 AND #I THEN
       #CMD.Start_A := TRUE;
       #CMD.Start_A := FALSE;
   END_IF;
END_REGION

REGION Network 3: Фильтр дребезга наличия сигнала
   RUNG wire#powerrail
      Contact( #CMD.Start_A )
      Coil( #Filter_On.Start )
      wire#w1
      Contact( #Filter_On."Exit" )
      S_Coil( #Data )
   END_RUNG
   RUNG wire#w1
      I_Contact( #Filter_On."Exit" )
      R_Coil( #Data )
   END_RUNG
   // the same network as SCL:
   #Filter_On.Start := #CMD.Start_A;
   IF #CMD.Start_A AND #Filter_On."Exit" THEN #Data := TRUE; END_IF;
   IF #CMD.Start_A AND NOT #Filter_On."Exit" THEN #Data := FALSE; END_IF;
END_REGION

REGION Network 4: Фильтр дребезга отсутствия сигнала
   RUNG wire#powerrail
      I_Contact( #CMD.Start_A )
      Coil( #Filter_Off.Start )
      wire#w1
      Contact( #Filter_Off."Exit" )
      R_Coil( #Data )
   END_RUNG
   RUNG wire#w1
      I_Contact( #Filter_Off."Exit" )
      S_Coil( #Data )
   END_RUNG
   // the same network as SCL:
   #Filter_Off.Start := NOT #CMD.Start_A;
   IF NOT #CMD.Start_A AND #Filter_Off."Exit" THEN #Data := FALSE; END_IF;
   IF NOT #CMD.Start_A AND NOT #Filter_Off."Exit" THEN #Data := TRUE; END_IF;
END_REGION

REGION Network 5: Блок таймеров
   RUNG wire#powerrail
      #Filter_On()
      #Filter_Off()
   END_RUNG
   // the same network as SCL:
   #Filter_On(ENO => #_w1);   // "Time_S_b"
   IF #_w1 THEN
       #Filter_Off();   // "Time_S_b"
   END_IF;
END_REGION

REGION Network 6: Управление запуском
   RUNG wire#powerrail
      Contact( #Data )
      I_Contact( #Use.Inverse )
      wire#w1
      I_Contact( #CMD.Hand )
      wire#w2
      S_SR(operand := #CMD.Start_M, r1 := wire#w4)
      Coil( #Signal )
   END_RUNG
   RUNG wire#powerrail
      I_Contact( #Data )
      Contact( #Use.Inverse )
   END_RUNG wire#w1
   RUNG wire#powerrail
      Contact( #CMD.Hand )
      Contact( #CMD.Start_M )
   END_RUNG wire#w2
   RUNG wire#powerrail
      Contact( #Data )
      Contact( #Use.Inverse )
      wire#w3
      I_Contact( #CMD.Hand )
   END_RUNG wire#w4
   RUNG wire#powerrail
      I_Contact( #Data )
      I_Contact( #Use.Inverse )
   END_RUNG wire#w3
   RUNG wire#powerrail
      Contact( #CMD.Hand )
      I_Contact( #CMD.Start_M )
   END_RUNG wire#w4
   // the same network as SCL:
   #_w1 := (((#Data AND #Use.Inverse) OR (NOT #Data AND NOT #Use.Inverse)) AND NOT #CMD.Hand) OR (#CMD.Hand AND NOT #CMD.Start_M);
   IF (((#Data AND NOT #Use.Inverse) OR (NOT #Data AND #Use.Inverse)) AND NOT #CMD.Hand) OR (#CMD.Hand AND #CMD.Start_M) THEN
       #CMD.Start_M := TRUE;   // SR flip-flop
   END_IF;
   IF #_w1 THEN #CMD.Start_M := FALSE; END_IF;
   #Signal := #CMD.Start_M;
END_REGION
END_FUNCTION_BLOCK

FUNCTION_BLOCK "Time_S_b"   // FB89, LAD
{ S7_Optimized_Access := 'FALSE' }
VERSION : 0.1
// stored: AutoNumber false, IsIECCheckEnabled false, SetENOAutomatically false, UDAEnableTagReadback false
   VAR DB_SPECIFIC
      SP { S7_SetPoint := 'True'} : Byte := 2;   // Уставка
      Now : Byte;   // Текущий счёт
      Start : Bool;   // Запуск
      "Exit" : Bool;   // Счёт завершён
      Pause : Bool;   // Пауза
      Reset : Bool;   // Сброс таймера
   END_VAR
   VAR_TEMP   // added for the SCL form of the ladder/FBD networks
      _w1 : Bool;
   END_VAR
BEGIN

REGION Network 1: Подсчёт времени
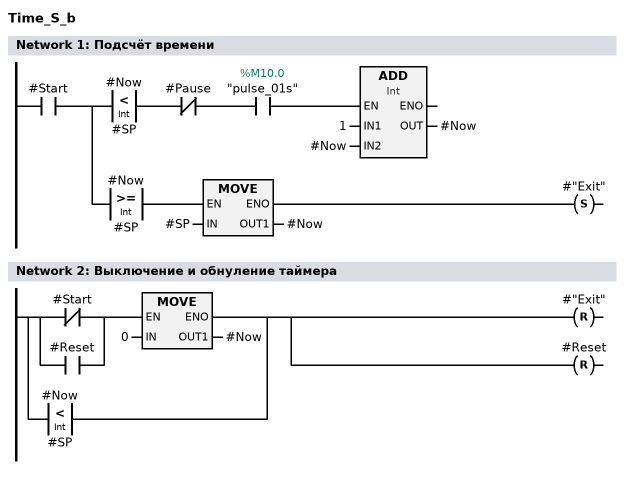
   RUNG wire#powerrail
      Contact( #Start )
      wire#w1
      { S7_Templates := "SrcType := Int" } LT_Contact(in1 := #Now, in2 := #SP)
      I_Contact( #Pause )
      Contact( "pulse_01s" )
      { S7_Templates := "SrcType := Int"; S7_GenerateENO := "TRUE" } Add(in1 := 1, in2 := #Now, out => #Now)
   END_RUNG
   RUNG wire#w1
      { S7_Templates := "SrcType := Int" } GE_Contact(in1 := #Now, in2 := #SP)
      { S7_GenerateENO := "TRUE" } Move(in := #SP, out1 => #Now)
      S_Coil( #"Exit" )
   END_RUNG
   // the same network as SCL:
   // ENO of a box is taken as its EN; it also drops when the box reports an error
   IF #Start AND (#Now < #SP) AND NOT #Pause AND "pulse_01s" THEN #Now := 1 + #Now; END_IF;
   #_w1 := #Start AND (#Now >= #SP);
   IF #_w1 THEN
       #Now := #SP;
       #"Exit" := TRUE;
   END_IF;
END_REGION

REGION Network 2: Выключение и обнуление таймера
   RUNG wire#powerrail
      I_Contact( #Start )
      wire#w1
      { S7_GenerateENO := "TRUE" } Move(in := 0, out1 => #Now)
      wire#w2
      R_Coil( #"Exit" )
   END_RUNG
   RUNG wire#powerrail
      Contact( #Reset )
   END_RUNG wire#w1
   RUNG wire#powerrail
      { S7_Templates := "SrcType := Int" } LT_Contact(in1 := #Now, in2 := #SP)
   END_RUNG wire#w2
   RUNG wire#w2
      R_Coil( #Reset )
   END_RUNG
   // the same network as SCL:
   // ENO of a box is taken as its EN; it also drops when the box reports an error
   #_w1 := NOT #Start OR #Reset;
   IF #_w1 THEN #Now := 0; END_IF;
   IF #_w1 OR (#Now < #SP) THEN
       #"Exit" := FALSE;
       #Reset := FALSE;
   END_IF;
END_REGION
END_FUNCTION_BLOCK

FUNCTION_BLOCK "AIx"   // FB220, LAD
{ S7_Optimized_Access := 'FALSE' }
VERSION : 0.1
// Signal - PIW код сигнала от датчика
// pulse - частота алгоритма фильтрации
// Result - результат обработки сигнала, формат Real
// stored: AutoNumber false, IsIECCheckEnabled false, SetENOAutomatically false, UDAEnableTagReadback false
   VAR DB_SPECIFIC
      Time_DTL { S7_SetPoint := 'True'} : DTL;
   END_VAR
   VAR_TEMP   // added for the SCL form of the ladder/FBD networks
      _w1 : Bool;
   END_VAR
BEGIN

REGION Network 1: Датчик уровня
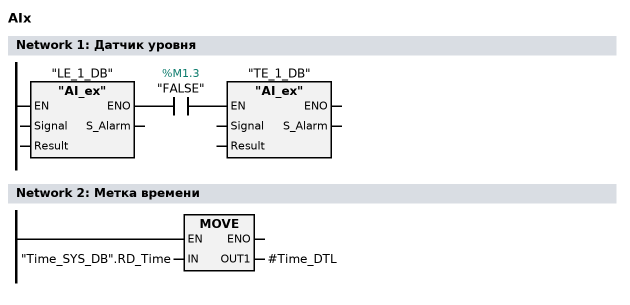
   RUNG wire#powerrail
      "LE_1_DB"(Signal :=, Result :=, S_Alarm =>)
      Contact( "FALSE" )
      "TE_1_DB"(Signal :=, Result :=, S_Alarm =>)
   END_RUNG
   // the same network as SCL:
   "LE_1_DB"(ENO => #_w1);   // "AI_ex"
   IF #_w1 AND "FALSE" THEN
       "TE_1_DB"();   // "AI_ex"
   END_IF;
END_REGION

REGION Network 2: Метка времени
   RUNG wire#powerrail
      Move(in := "Time_SYS_DB".RD_Time, out1 => #Time_DTL)
   END_RUNG
   // the same network as SCL:
   #Time_DTL := "Time_SYS_DB".RD_Time;
END_REGION
END_FUNCTION_BLOCK

FUNCTION_BLOCK "AI_ex"   // FB103, LAD
{ S7_Optimized_Access := 'FALSE' }
VERSION : 0.1
// stored: AutoNumber false, IsIECCheckEnabled false, SetENOAutomatically false, UDAEnableTagReadback false
   VAR_OUTPUT
      S_Alarm : Bool;   // Внешний индикатор наличия аварии
   END_VAR
   VAR_IN_OUT
      Signal : Int;   // Входной сигнал контроллера
      Result : Real;   // Результат измерений
   END_VAR
   VAR DB_SPECIFIC
      CMD : "CMD";   // Основные команды / Блок команд
      Mode : Int;   // Режим работы
      Status : Int;   // Статус устройства
      Use : Struct   // Функционал
         RTD { S7_SetPoint := 'True'} : Bool;   // Режим RTD
         Filter { S7_SetPoint := 'True'} : Bool;   // Филтрация сигнала
         Inverse { S7_SetPoint := 'True'} : Bool;   // Инверсия сигнала
         Indirect { S7_SetPoint := 'True'} : Bool := true;   // Косвенная адресация
         Status { S7_SetPoint := 'True'} : Bool;   // Использовать подсветку
         Light : Bool;   // Динамическая подсветка
         Lim_Low : Bool;   // Отсечь низкие аварии
         Lim_High : Bool;   // Отсечь высокие аварии
         Communication { S7_SetPoint := 'True'} : Bool;   // Передача в Value по сети
      END_STRUCT;
      VmA : Real;   // Реальный сигнал на входе ПЛК
      RTD_c { S7_SetPoint := 'True'} : Real := 10.0;   // Коэффициент RTD
      Calibration { S7_SetPoint := 'True'} : Real;   // Поправка
   END_VAR
   VAR
      Converter { S7_SetPoint := 'True'} : "Converter";   // Масштабирование сигнала
   END_VAR
   VAR DB_SPECIFIC
      SP : Struct   // Уставки аварий
         NC { S7_SetPoint := 'True'} : Real := -500.0;   // Сигнал при обрыве линии
         SC { S7_SetPoint := 'True'} : Real := 32000.0;   // Сигнал при КЗ/перегрузке
         HH { S7_SetPoint := 'True'} : Real := 90.0;   // Аварийно высокий сигнал
         H { S7_SetPoint := 'True'} : Real := 85.0;   // Высокий сигнал
         L { S7_SetPoint := 'True'} : Real := 15.0;   // Низкий сигнал
         LL { S7_SetPoint := 'True'} : Real := 10.0;   // Аварийно низкий сигнал
      END_STRUCT;
   END_VAR
   VAR
      Tx { S7_SetPoint := 'True'} : Array[0..5] of "Time_R";   // Блок таймеров
   END_VAR
   VAR DB_SPECIFIC
      Alarm : Struct   // Список аварий
         ST : Bool;   // Общая неисправность
         HH : Bool;   // сработала авария по аварийно высокму уровню
         H : Bool;   // сработало предупреждение по высокому уровню
         L : Bool;   // сработало предупреждение по низкому уровню
         LL : Bool;   // сработало предупрждение по аварийно низкому уровню
         NC : Bool;   // обрыв линии
         SC : Bool;   // короткое замыкание
      END_STRUCT;
      Alarms : Word;   // Слово аварий
      Events : Word;   // События датчика
      pos : Array[0..15] of Bool;   // Контроль фронтов событий
      Input_Type { S7_SetPoint := 'True'} : Int;   // Тип датчика, 0 - 4..20, 1 - 0..20, 2 - 0..10, 3 - 0..5, 4 - RTD
      CodeID { S7_SetPoint := 'True'} : Int;   // Код датчика для привязки в скаде
      "Type" { S7_SetPoint := 'True'} : Int;   // Тип датчика (единицы измерения)
      ADDR { S7_SetPoint := 'True'} : Int;   // Адрес входа на контроллере
      Filter_SP { S7_SetPoint := 'True'} : Int := 100;   // Ёмкость фильтра
   END_VAR
   VAR
      Filter_DB : "Filter";   // Фильтрация скачков сигнала
   END_VAR
   VAR DB_SPECIFIC
      Time_DTL { S7_SetPoint := 'True'} : DTL;
   END_VAR
   VAR_TEMP
      ev : Bool;   // Флаг событий
      Value : Real;   // Итоговый сигнал
      Signal_DI : DInt;   // Конвертация сигнала
      Signal_R : Real;   // Конвертация сигнала
      Type_Min : Real;
      Type_Max : Real;
   END_VAR
   VAR CONSTANT
      FALSE : Bool;
      TRUE : Bool := true;
   END_VAR
   // CMD.Start_A := true;
   // Converter.Max_In := 27648.0;
   // Converter.Max_Out := 100.0;
   VAR_TEMP   // added for the SCL form of the ladder/FBD networks
      _w1 : Bool;
      _w2 : Bool;
      _w3 : Bool;
      _w4 : Bool;
      _w5 : Bool;
      _w6 : Bool;
      _w7 : Bool;
      _w8 : Bool;
      _w9 : Bool;
      _w10 : Bool;
      _w11 : Bool;
      _w12 : Bool;
      _w13 : Bool;
      _w14 : Bool;
      _w15 : Bool;
      _w16 : Bool;
   END_VAR
BEGIN

REGION Network 1: Общий сброс
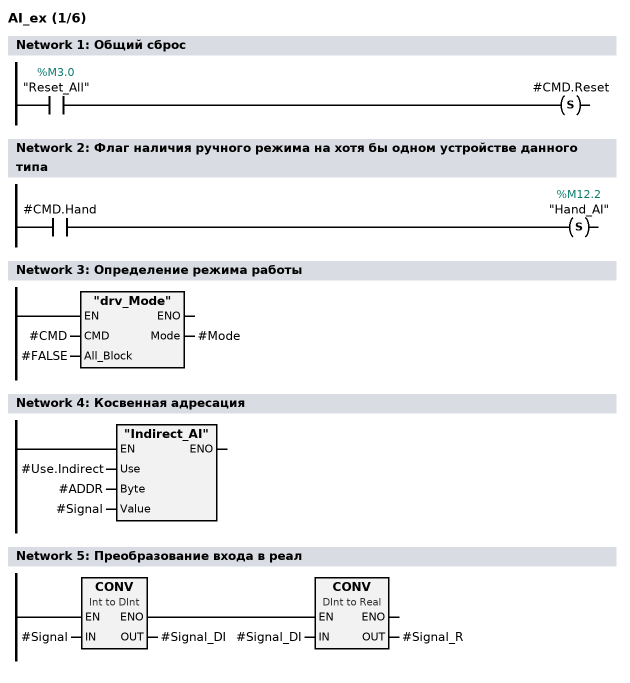
   RUNG wire#powerrail
      Contact( "Reset_All" )
      S_Coil( #CMD.Reset )
   END_RUNG
   // the same network as SCL:
   IF "Reset_All" THEN #CMD.Reset := TRUE; END_IF;
END_REGION

REGION Network 2: Флаг наличия ручного режима на хотя бы одном устройстве данного типа
   RUNG wire#powerrail
      Contact( #CMD.Hand )
      S_Coil( "Hand_AI" )
   END_RUNG
   // the same network as SCL:
   IF #CMD.Hand THEN "Hand_AI" := TRUE; END_IF;
END_REGION

REGION Network 3: Определение режима работы
   RUNG wire#powerrail
      "drv_Mode"(CMD := #CMD, All_Block := #FALSE, Mode => #Mode)
   END_RUNG
   // the same network as SCL:
   "drv_Mode"(CMD := #CMD, All_Block := #FALSE, Mode => #Mode);
END_REGION

REGION Network 4: Косвенная адресация
   RUNG wire#powerrail
      "Indirect_AI"(Use := #Use.Indirect, "Byte" := #ADDR, Value := #Signal)
   END_RUNG
   // the same network as SCL:
   "Indirect_AI"(Use := #Use.Indirect, "Byte" := #ADDR, Value := #Signal);
END_REGION

REGION Network 5: Преобразование входа в реал
   RUNG wire#powerrail
      { S7_Templates := "[SrcType := Int, DestType := DInt]"; S7_GenerateENO := "TRUE" } Convert(in := #Signal, out => #Signal_DI)
      { S7_Templates := "[SrcType := DInt, DestType := Real]"; S7_GenerateENO := "TRUE" } Convert(in := #Signal_DI, out => #Signal_R)
   END_RUNG
   // the same network as SCL:
   // ENO of a box is taken as its EN; it also drops when the box reports an error
   #Signal_DI := INT_TO_DINT(#Signal);
   #Signal_R := DINT_TO_REAL(#Signal_DI);
END_REGION

REGION Network 6: Преобразование кода в реальное значение входа
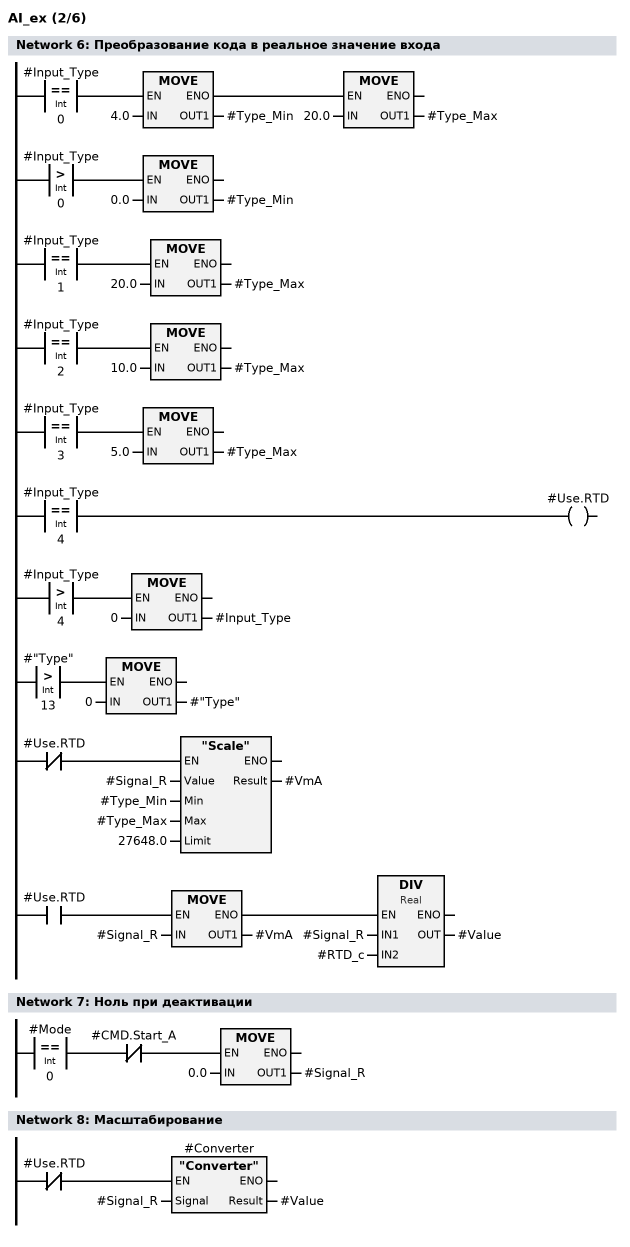
   RUNG wire#powerrail
      { S7_Templates := "SrcType := Int" } EQ_Contact(in1 := #Input_Type, in2 := 0)
      Move(in := 4.0, out1 => #Type_Min)
      Move(in := 20.0, out1 => #Type_Max)
   END_RUNG
   RUNG wire#powerrail
      { S7_Templates := "SrcType := Int" } GT_Contact(in1 := #Input_Type, in2 := 0)
      Move(in := 0.0, out1 => #Type_Min)
   END_RUNG
   RUNG wire#powerrail
      { S7_Templates := "SrcType := Int" } EQ_Contact(in1 := #Input_Type, in2 := 1)
      Move(in := 20.0, out1 => #Type_Max)
   END_RUNG
   RUNG wire#powerrail
      { S7_Templates := "SrcType := Int" } EQ_Contact(in1 := #Input_Type, in2 := 2)
      Move(in := 10.0, out1 => #Type_Max)
   END_RUNG
   RUNG wire#powerrail
      { S7_Templates := "SrcType := Int" } EQ_Contact(in1 := #Input_Type, in2 := 3)
      Move(in := 5.0, out1 => #Type_Max)
   END_RUNG
   RUNG wire#powerrail
      { S7_Templates := "SrcType := Int" } EQ_Contact(in1 := #Input_Type, in2 := 4)
      Coil( #Use.RTD )
   END_RUNG
   RUNG wire#powerrail
      { S7_Templates := "SrcType := Int" } GT_Contact(in1 := #Input_Type, in2 := 4)
      Move(in := 0, out1 => #Input_Type)
   END_RUNG
   RUNG wire#powerrail
      { S7_Templates := "SrcType := Int" } GT_Contact(in1 := #"Type", in2 := 13)
      Move(in := 0, out1 => #"Type")
   END_RUNG
   RUNG wire#powerrail
      I_Contact( #Use.RTD )
      "Scale"(Value := #Signal_R, Min := #Type_Min, Max := #Type_Max, Limit := 27648.0, Result => #VmA)
   END_RUNG
   RUNG wire#powerrail
      Contact( #Use.RTD )
      Move(in := #Signal_R, out1 => #VmA)
      { S7_Templates := "SrcType := Real"; S7_GenerateENO := "TRUE" } Div(in1 := #Signal_R, in2 := #RTD_c, out => #Value)
   END_RUNG
   // the same network as SCL:
   IF #Input_Type = 0 THEN
       #Type_Min := 4.0;
       #Type_Max := 20.0;
   END_IF;
   IF #Input_Type > 0 THEN #Type_Min := 0.0; END_IF;
   IF #Input_Type = 1 THEN #Type_Max := 20.0; END_IF;
   IF #Input_Type = 2 THEN #Type_Max := 10.0; END_IF;
   IF #Input_Type = 3 THEN #Type_Max := 5.0; END_IF;
   #Use.RTD := #Input_Type = 4;
   IF #Input_Type > 4 THEN #Input_Type := 0; END_IF;
   IF #"Type" > 13 THEN #"Type" := 0; END_IF;
   IF NOT #Use.RTD THEN
       "Scale"(Value := #Signal_R, Min := #Type_Min, Max := #Type_Max, Limit := 27648.0, Result => #VmA);
   END_IF;
   IF #Use.RTD THEN
       #VmA := #Signal_R;
       #Value := #Signal_R / #RTD_c;
   END_IF;
END_REGION

REGION Network 7: Ноль при деактивации
   RUNG wire#powerrail
      { S7_Templates := "SrcType := Int" } EQ_Contact(in1 := #Mode, in2 := 0)
      I_Contact( #CMD.Start_A )
      Move(in := 0.0, out1 => #Signal_R)
   END_RUNG
   // the same network as SCL:
   IF (#Mode = 0) AND NOT #CMD.Start_A THEN #Signal_R := 0.0; END_IF;
END_REGION

REGION Network 8: Масштабирование
   RUNG wire#powerrail
      I_Contact( #Use.RTD )
      #Converter(Signal := #Signal_R, Result => #Value)
   END_RUNG
   // the same network as SCL:
   IF NOT #Use.RTD THEN
       #Converter(Signal := #Signal_R, Result => #Value);   // "Converter"
   END_IF;
END_REGION

REGION Network 9: Вызов блока фильтрации
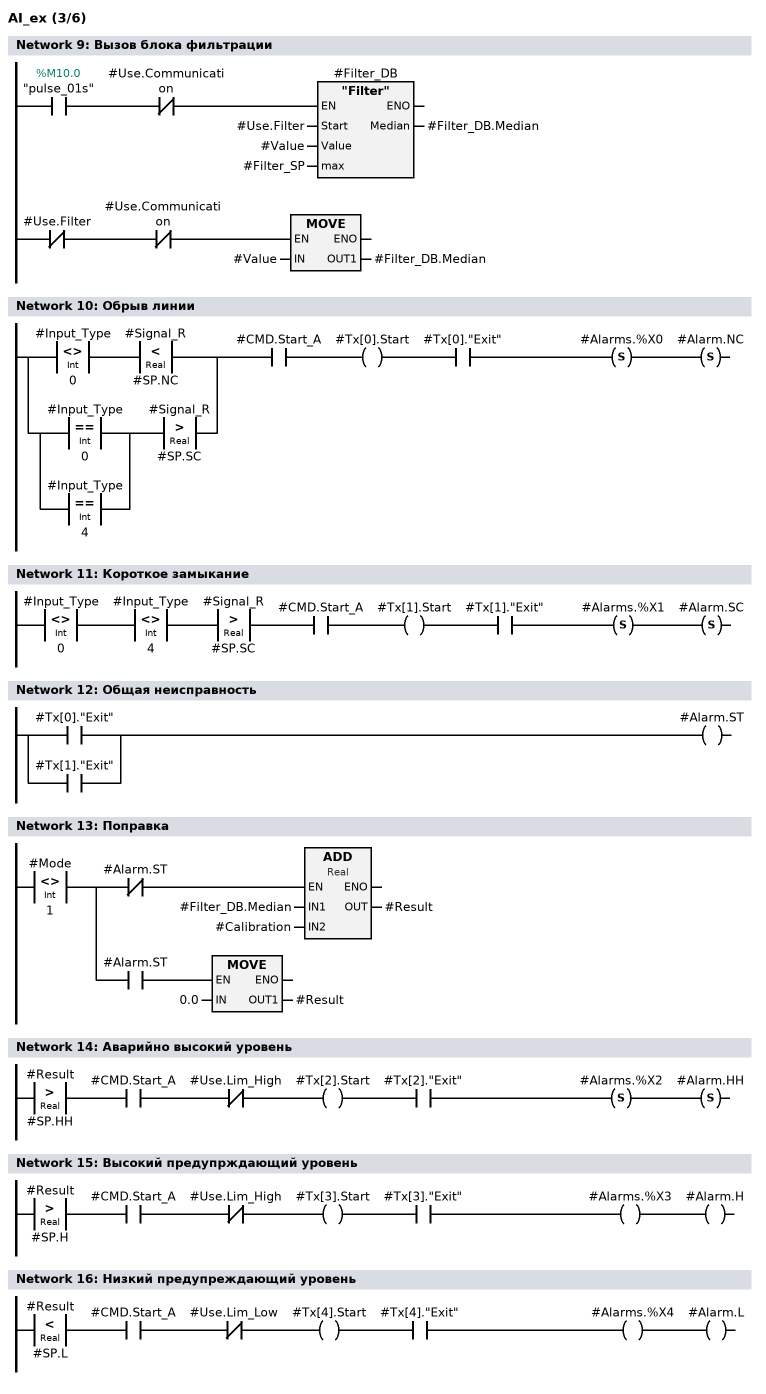
   RUNG wire#powerrail
      Contact( "pulse_01s" )
      I_Contact( #Use.Communication )
      #Filter_DB(Start := #Use.Filter, Value := #Value, max := #Filter_SP, Median => #Filter_DB.Median)
   END_RUNG
   RUNG wire#powerrail
      I_Contact( #Use.Filter )
      I_Contact( #Use.Communication )
      { S7_GenerateENO := "TRUE" } Move(in := #Value, out1 => #Filter_DB.Median)
   END_RUNG
   // the same network as SCL:
   IF "pulse_01s" AND NOT #Use.Communication THEN
       #Filter_DB(Start := #Use.Filter, Value := #Value, max := #Filter_SP, Median => #Filter_DB.Median);   // "Filter"
   END_IF;
   IF NOT #Use.Filter AND NOT #Use.Communication THEN #Filter_DB.Median := #Value; END_IF;
END_REGION

REGION Network 10: Обрыв линии
   RUNG wire#powerrail
      { S7_Templates := "SrcType := Int" } NE_Contact(in1 := #Input_Type, in2 := 0)
      { S7_Templates := "SrcType := Real" } LT_Contact(in1 := #Signal_R, in2 := #SP.NC)
      wire#w1
      Contact( #CMD.Start_A )
      Coil( #Tx[0].Start )
      Contact( #Tx[0]."Exit" )
      S_Coil( #Alarms.%X0 )
      S_Coil( #Alarm.NC )
   END_RUNG
   RUNG wire#powerrail
      { S7_Templates := "SrcType := Int" } EQ_Contact(in1 := #Input_Type, in2 := 0)
      wire#w2
      { S7_Templates := "SrcType := Real" } GT_Contact(in1 := #Signal_R, in2 := #SP.SC)
   END_RUNG wire#w1
   RUNG wire#powerrail
      { S7_Templates := "SrcType := Int" } EQ_Contact(in1 := #Input_Type, in2 := 4)
   END_RUNG wire#w2
   // the same network as SCL:
   #Tx[0].Start := (((#Input_Type <> 0) AND (#Signal_R < #SP.NC)) OR (((#Input_Type = 0) OR (#Input_Type = 4)) AND (#Signal_R > #SP.SC))) AND #CMD.Start_A;
   IF (((#Input_Type <> 0) AND (#Signal_R < #SP.NC)) OR (((#Input_Type = 0) OR (#Input_Type = 4)) AND (#Signal_R > #SP.SC))) AND #CMD.Start_A AND #Tx[0]."Exit" THEN
       #Alarms.%X0 := TRUE;
       #Alarm.NC := TRUE;
   END_IF;
END_REGION

REGION Network 11: Короткое замыкание
   RUNG wire#powerrail
      { S7_Templates := "SrcType := Int" } NE_Contact(in1 := #Input_Type, in2 := 0)
      { S7_Templates := "SrcType := Int" } NE_Contact(in1 := #Input_Type, in2 := 4)
      { S7_Templates := "SrcType := Real" } GT_Contact(in1 := #Signal_R, in2 := #SP.SC)
      Contact( #CMD.Start_A )
      Coil( #Tx[1].Start )
      Contact( #Tx[1]."Exit" )
      S_Coil( #Alarms.%X1 )
      S_Coil( #Alarm.SC )
   END_RUNG
   // the same network as SCL:
   #Tx[1].Start := (#Input_Type <> 0) AND (#Input_Type <> 4) AND (#Signal_R > #SP.SC) AND #CMD.Start_A;
   IF (#Input_Type <> 0) AND (#Input_Type <> 4) AND (#Signal_R > #SP.SC) AND #CMD.Start_A AND #Tx[1]."Exit" THEN
       #Alarms.%X1 := TRUE;
       #Alarm.SC := TRUE;
   END_IF;
END_REGION

REGION Network 12: Общая неисправность
   RUNG wire#powerrail
      Contact( #Tx[0]."Exit" )
      wire#w1
      Coil( #Alarm.ST )
   END_RUNG
   RUNG wire#powerrail
      Contact( #Tx[1]."Exit" )
   END_RUNG wire#w1
   // the same network as SCL:
   #Alarm.ST := #Tx[0]."Exit" OR #Tx[1]."Exit";
END_REGION

REGION Network 13: Поправка
   RUNG wire#powerrail
      { S7_Templates := "SrcType := Int" } NE_Contact(in1 := #Mode, in2 := 1)
      wire#w1
      I_Contact( #Alarm.ST )
      { S7_Templates := "SrcType := Real"; S7_GenerateENO := "TRUE" } Add(in1 := #Filter_DB.Median, in2 := #Calibration, out => #Result)
   END_RUNG
   RUNG wire#w1
      Contact( #Alarm.ST )
      Move(in := 0.0, out1 => #Result)
   END_RUNG
   // the same network as SCL:
   #_w1 := #Mode <> 1;
   IF #_w1 AND NOT #Alarm.ST THEN #Result := #Filter_DB.Median + #Calibration; END_IF;
   IF #_w1 AND #Alarm.ST THEN #Result := 0.0; END_IF;
END_REGION

REGION Network 14: Аварийно высокий уровень
   RUNG wire#powerrail
      { S7_Templates := "SrcType := Real" } GT_Contact(in1 := #Result, in2 := #SP.HH)
      Contact( #CMD.Start_A )
      I_Contact( #Use.Lim_High )
      Coil( #Tx[2].Start )
      Contact( #Tx[2]."Exit" )
      S_Coil( #Alarms.%X2 )
      S_Coil( #Alarm.HH )
   END_RUNG
   // the same network as SCL:
   #Tx[2].Start := (#Result > #SP.HH) AND #CMD.Start_A AND NOT #Use.Lim_High;
   IF (#Result > #SP.HH) AND #CMD.Start_A AND NOT #Use.Lim_High AND #Tx[2]."Exit" THEN
       #Alarms.%X2 := TRUE;
       #Alarm.HH := TRUE;
   END_IF;
END_REGION

REGION Network 15: Высокий предупрждающий уровень
   RUNG wire#powerrail
      { S7_Templates := "SrcType := Real" } GT_Contact(in1 := #Result, in2 := #SP.H)
      Contact( #CMD.Start_A )
      I_Contact( #Use.Lim_High )
      Coil( #Tx[3].Start )
      Contact( #Tx[3]."Exit" )
      Coil( #Alarms.%X3 )
      Coil( #Alarm.H )
   END_RUNG
   // the same network as SCL:
   #Tx[3].Start := (#Result > #SP.H) AND #CMD.Start_A AND NOT #Use.Lim_High;
   #Alarms.%X3 := (#Result > #SP.H) AND #CMD.Start_A AND NOT #Use.Lim_High AND #Tx[3]."Exit";
   #Alarm.H := #Alarms.%X3;
END_REGION

REGION Network 16: Низкий предупреждающий уровень
   RUNG wire#powerrail
      { S7_Templates := "SrcType := Real" } LT_Contact(in1 := #Result, in2 := #SP.L)
      Contact( #CMD.Start_A )
      I_Contact( #Use.Lim_Low )
      Coil( #Tx[4].Start )
      Contact( #Tx[4]."Exit" )
      Coil( #Alarms.%X4 )
      Coil( #Alarm.L )
   END_RUNG
   // the same network as SCL:
   #Tx[4].Start := (#Result < #SP.L) AND #CMD.Start_A AND NOT #Use.Lim_Low;
   #Alarms.%X4 := (#Result < #SP.L) AND #CMD.Start_A AND NOT #Use.Lim_Low AND #Tx[4]."Exit";
   #Alarm.L := #Alarms.%X4;
END_REGION

REGION Network 17: Аварийно высокий уровень
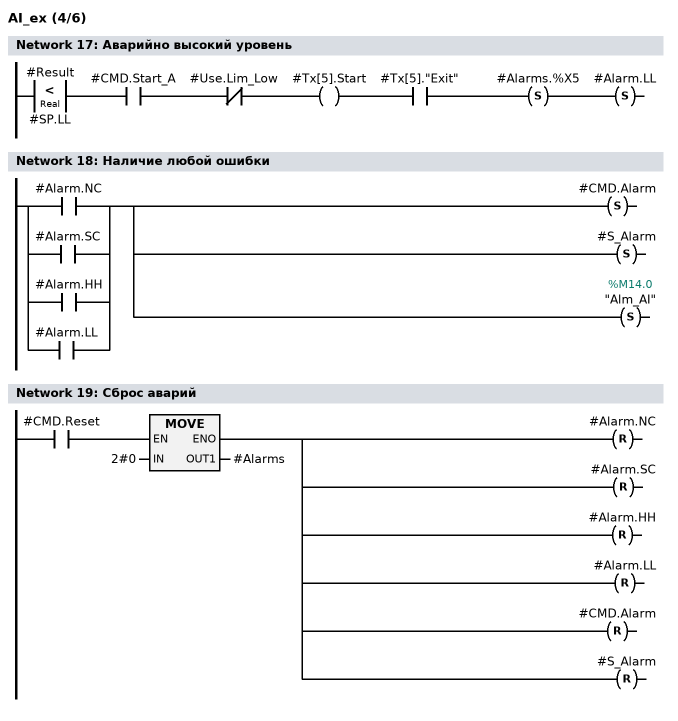
   RUNG wire#powerrail
      { S7_Templates := "SrcType := Real" } LT_Contact(in1 := #Result, in2 := #SP.LL)
      Contact( #CMD.Start_A )
      I_Contact( #Use.Lim_Low )
      Coil( #Tx[5].Start )
      Contact( #Tx[5]."Exit" )
      S_Coil( #Alarms.%X5 )
      S_Coil( #Alarm.LL )
   END_RUNG
   // the same network as SCL:
   #Tx[5].Start := (#Result < #SP.LL) AND #CMD.Start_A AND NOT #Use.Lim_Low;
   IF (#Result < #SP.LL) AND #CMD.Start_A AND NOT #Use.Lim_Low AND #Tx[5]."Exit" THEN
       #Alarms.%X5 := TRUE;
       #Alarm.LL := TRUE;
   END_IF;
END_REGION

REGION Network 18: Наличие любой ошибки
   RUNG wire#powerrail
      Contact( #Alarm.NC )
      wire#w1
      S_Coil( #CMD.Alarm )
   END_RUNG
   RUNG wire#powerrail
      Contact( #Alarm.SC )
   END_RUNG wire#w1
   RUNG wire#powerrail
      Contact( #Alarm.HH )
   END_RUNG wire#w1
   RUNG wire#powerrail
      Contact( #Alarm.LL )
   END_RUNG wire#w1
   RUNG wire#w1
      S_Coil( #S_Alarm )
   END_RUNG
   RUNG wire#w1
      S_Coil( "Alm_AI" )
   END_RUNG
   // the same network as SCL:
   IF #Alarm.NC OR #Alarm.SC OR #Alarm.HH OR #Alarm.LL THEN
       #CMD.Alarm := TRUE;
       #S_Alarm := TRUE;
       "Alm_AI" := TRUE;
   END_IF;
END_REGION

REGION Network 19: Сброс аварий
   RUNG wire#powerrail
      Contact( #CMD.Reset )
      Move(in := 2#0, out1 => #Alarms)
      wire#w1
      R_Coil( #Alarm.NC )
   END_RUNG
   RUNG wire#w1
      R_Coil( #Alarm.SC )
   END_RUNG
   RUNG wire#w1
      R_Coil( #Alarm.HH )
   END_RUNG
   RUNG wire#w1
      R_Coil( #Alarm.LL )
   END_RUNG
   RUNG wire#w1
      R_Coil( #CMD.Alarm )
   END_RUNG
   RUNG wire#w1
      R_Coil( #S_Alarm )
   END_RUNG
   // the same network as SCL:
   IF #CMD.Reset THEN
       #Alarms := 2#0;
       #Alarm.NC := FALSE;
       #Alarm.SC := FALSE;
       #Alarm.HH := FALSE;
       #Alarm.LL := FALSE;
       #CMD.Alarm := FALSE;
       #S_Alarm := FALSE;
   END_IF;
END_REGION

REGION Network 20: События датчика
   // 0 - датчик активирован
   // 1 - датчик деактивирован
   // 2 - датчик в ручном режиме
   // 3 - датчик в автоматическом режиме
   // 4 - сигнал ниже нижнего предупреждающего
   // 5 - сигнал в норме
   // 6 - сигнал выше верхнего предупреждающего
   // 7 - сигнал в норме
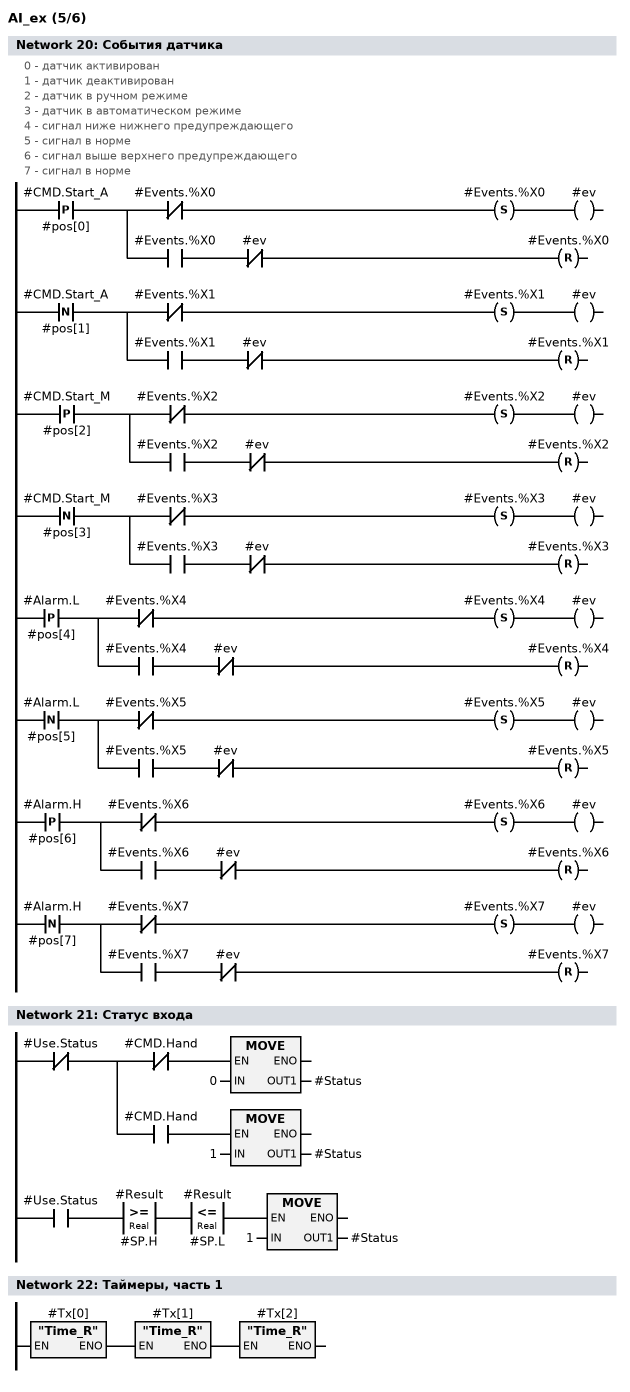
   RUNG wire#powerrail
      P_Contact(operand := #CMD.Start_A, bit := #pos[0])
      wire#w1
      I_Contact( #Events.%X0 )
      S_Coil( #Events.%X0 )
      Coil( #ev )
   END_RUNG
   RUNG wire#w1
      Contact( #Events.%X0 )
      I_Contact( #ev )
      R_Coil( #Events.%X0 )
   END_RUNG
   RUNG wire#powerrail
      N_Contact(operand := #CMD.Start_A, bit := #pos[1])
      wire#w2
      I_Contact( #Events.%X1 )
      S_Coil( #Events.%X1 )
      Coil( #ev )
   END_RUNG
   RUNG wire#w2
      Contact( #Events.%X1 )
      I_Contact( #ev )
      R_Coil( #Events.%X1 )
   END_RUNG
   RUNG wire#powerrail
      P_Contact(operand := #CMD.Start_M, bit := #pos[2])
      wire#w3
      I_Contact( #Events.%X2 )
      S_Coil( #Events.%X2 )
      Coil( #ev )
   END_RUNG
   RUNG wire#w3
      Contact( #Events.%X2 )
      I_Contact( #ev )
      R_Coil( #Events.%X2 )
   END_RUNG
   RUNG wire#powerrail
      N_Contact(operand := #CMD.Start_M, bit := #pos[3])
      wire#w4
      I_Contact( #Events.%X3 )
      S_Coil( #Events.%X3 )
      Coil( #ev )
   END_RUNG
   RUNG wire#w4
      Contact( #Events.%X3 )
      I_Contact( #ev )
      R_Coil( #Events.%X3 )
   END_RUNG
   RUNG wire#powerrail
      P_Contact(operand := #Alarm.L, bit := #pos[4])
      wire#w5
      I_Contact( #Events.%X4 )
      S_Coil( #Events.%X4 )
      Coil( #ev )
   END_RUNG
   RUNG wire#w5
      Contact( #Events.%X4 )
      I_Contact( #ev )
      R_Coil( #Events.%X4 )
   END_RUNG
   RUNG wire#powerrail
      N_Contact(operand := #Alarm.L, bit := #pos[5])
      wire#w6
      I_Contact( #Events.%X5 )
      S_Coil( #Events.%X5 )
      Coil( #ev )
   END_RUNG
   RUNG wire#w6
      Contact( #Events.%X5 )
      I_Contact( #ev )
      R_Coil( #Events.%X5 )
   END_RUNG
   RUNG wire#powerrail
      P_Contact(operand := #Alarm.H, bit := #pos[6])
      wire#w7
      I_Contact( #Events.%X6 )
      S_Coil( #Events.%X6 )
      Coil( #ev )
   END_RUNG
   RUNG wire#w7
      Contact( #Events.%X6 )
      I_Contact( #ev )
      R_Coil( #Events.%X6 )
   END_RUNG
   RUNG wire#powerrail
      N_Contact(operand := #Alarm.H, bit := #pos[7])
      wire#w8
      I_Contact( #Events.%X7 )
      S_Coil( #Events.%X7 )
      Coil( #ev )
   END_RUNG
   RUNG wire#w8
      Contact( #Events.%X7 )
      I_Contact( #ev )
      R_Coil( #Events.%X7 )
   END_RUNG
   // the same network as SCL:
   #_w1 := #CMD.Start_A AND NOT #pos[0];   // rising edge of #CMD.Start_A
   #pos[0] := #CMD.Start_A;
   #_w2 := #_w1 AND NOT #Events.%X0;
   IF #_w2 THEN #Events.%X0 := TRUE; END_IF;
   #ev := #_w2;
   IF #_w1 AND #Events.%X0 AND NOT #ev THEN #Events.%X0 := FALSE; END_IF;
   #_w3 := NOT #CMD.Start_A AND #pos[1];   // falling edge of #CMD.Start_A
   #pos[1] := #CMD.Start_A;
   #_w4 := #_w3 AND NOT #Events.%X1;
   IF #_w4 THEN #Events.%X1 := TRUE; END_IF;
   #ev := #_w4;
   IF #_w3 AND #Events.%X1 AND NOT #ev THEN #Events.%X1 := FALSE; END_IF;
   #_w5 := #CMD.Start_M AND NOT #pos[2];   // rising edge of #CMD.Start_M
   #pos[2] := #CMD.Start_M;
   #_w6 := #_w5 AND NOT #Events.%X2;
   IF #_w6 THEN #Events.%X2 := TRUE; END_IF;
   #ev := #_w6;
   IF #_w5 AND #Events.%X2 AND NOT #ev THEN #Events.%X2 := FALSE; END_IF;
   #_w7 := NOT #CMD.Start_M AND #pos[3];   // falling edge of #CMD.Start_M
   #pos[3] := #CMD.Start_M;
   #_w8 := #_w7 AND NOT #Events.%X3;
   IF #_w8 THEN #Events.%X3 := TRUE; END_IF;
   #ev := #_w8;
   IF #_w7 AND #Events.%X3 AND NOT #ev THEN #Events.%X3 := FALSE; END_IF;
   #_w9 := #Alarm.L AND NOT #pos[4];   // rising edge of #Alarm.L
   #pos[4] := #Alarm.L;
   #_w10 := #_w9 AND NOT #Events.%X4;
   IF #_w10 THEN #Events.%X4 := TRUE; END_IF;
   #ev := #_w10;
   IF #_w9 AND #Events.%X4 AND NOT #ev THEN #Events.%X4 := FALSE; END_IF;
   #_w11 := NOT #Alarm.L AND #pos[5];   // falling edge of #Alarm.L
   #pos[5] := #Alarm.L;
   #_w12 := #_w11 AND NOT #Events.%X5;
   IF #_w12 THEN #Events.%X5 := TRUE; END_IF;
   #ev := #_w12;
   IF #_w11 AND #Events.%X5 AND NOT #ev THEN #Events.%X5 := FALSE; END_IF;
   #_w13 := #Alarm.H AND NOT #pos[6];   // rising edge of #Alarm.H
   #pos[6] := #Alarm.H;
   #_w14 := #_w13 AND NOT #Events.%X6;
   IF #_w14 THEN #Events.%X6 := TRUE; END_IF;
   #ev := #_w14;
   IF #_w13 AND #Events.%X6 AND NOT #ev THEN #Events.%X6 := FALSE; END_IF;
   #_w15 := NOT #Alarm.H AND #pos[7];   // falling edge of #Alarm.H
   #pos[7] := #Alarm.H;
   #_w16 := #_w15 AND NOT #Events.%X7;
   IF #_w16 THEN #Events.%X7 := TRUE; END_IF;
   #ev := #_w16;
   IF #_w15 AND #Events.%X7 AND NOT #ev THEN #Events.%X7 := FALSE; END_IF;
END_REGION

REGION Network 21: Статус входа
   RUNG wire#powerrail
      I_Contact( #Use.Status )
      wire#w1
      I_Contact( #CMD.Hand )
      Move(in := 0, out1 => #Status)
   END_RUNG
   RUNG wire#w1
      Contact( #CMD.Hand )
      Move(in := 1, out1 => #Status)
   END_RUNG
   RUNG wire#powerrail
      Contact( #Use.Status )
      { S7_Templates := "SrcType := Real" } GE_Contact(in1 := #Result, in2 := #SP.H)
      { S7_Templates := "SrcType := Real" } LE_Contact(in1 := #Result, in2 := #SP.L)
      Move(in := 1, out1 => #Status)
   END_RUNG
   // the same network as SCL:
   IF NOT #Use.Status AND NOT #CMD.Hand THEN #Status := 0; END_IF;
   IF NOT #Use.Status AND #CMD.Hand THEN #Status := 1; END_IF;
   IF #Use.Status AND (#Result >= #SP.H) AND (#Result <= #SP.L) THEN #Status := 1; END_IF;
END_REGION

REGION Network 22: Таймеры, часть 1
   RUNG wire#powerrail
      #Tx[0]()
      #Tx[1]()
      #Tx[2]()
   END_RUNG
   // the same network as SCL:
   #Tx[0](ENO => #_w1);   // "Time_R"
   #Tx[1](EN := #_w1, ENO => #_w2);   // "Time_R"
   IF #_w2 THEN
       #Tx[2]();   // "Time_R"
   END_IF;
END_REGION

REGION Network 23: Таймеры, часть 2
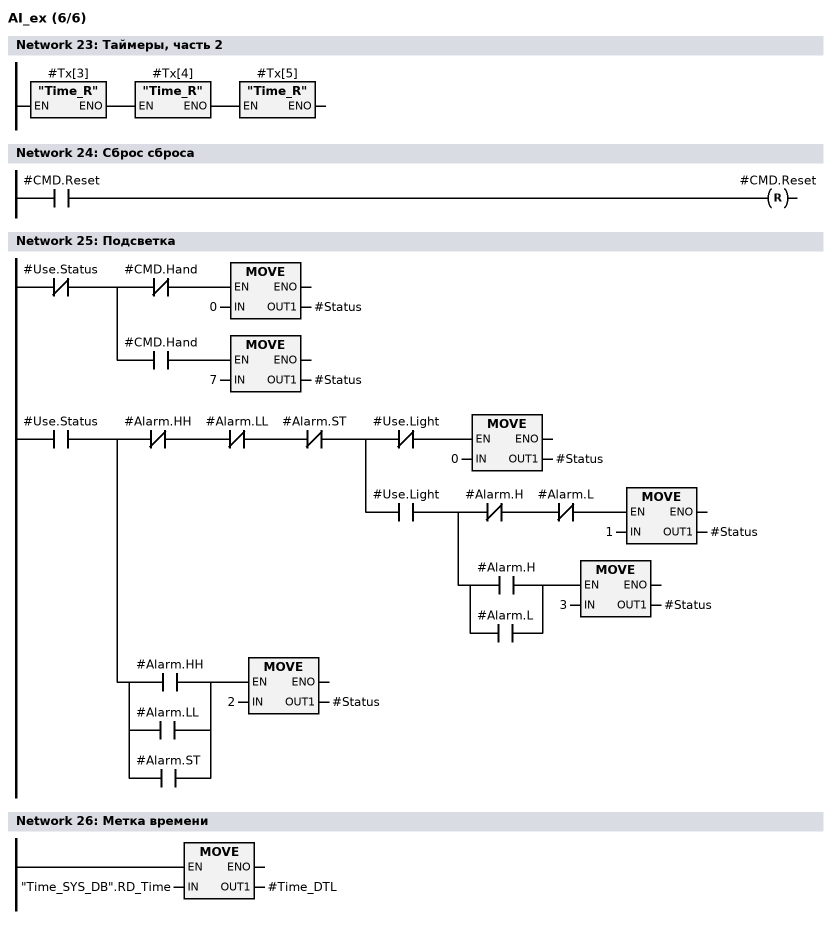
   RUNG wire#powerrail
      #Tx[3]()
      #Tx[4]()
      #Tx[5]()
   END_RUNG
   // the same network as SCL:
   #Tx[3](ENO => #_w1);   // "Time_R"
   #Tx[4](EN := #_w1, ENO => #_w2);   // "Time_R"
   IF #_w2 THEN
       #Tx[5]();   // "Time_R"
   END_IF;
END_REGION

REGION Network 24: Сброс сброса
   RUNG wire#powerrail
      Contact( #CMD.Reset )
      R_Coil( #CMD.Reset )
   END_RUNG
   // the same network as SCL:
   IF #CMD.Reset THEN #CMD.Reset := FALSE; END_IF;
END_REGION

REGION Network 25: Подсветка
   RUNG wire#powerrail
      I_Contact( #Use.Status )
      wire#w1
      I_Contact( #CMD.Hand )
      Move(in := 0, out1 => #Status)
   END_RUNG
   RUNG wire#w1
      Contact( #CMD.Hand )
      Move(in := 7, out1 => #Status)
   END_RUNG
   RUNG wire#powerrail
      Contact( #Use.Status )
      wire#w2
      I_Contact( #Alarm.HH )
      I_Contact( #Alarm.LL )
      I_Contact( #Alarm.ST )
      wire#w3
      I_Contact( #Use.Light )
      Move(in := 0, out1 => #Status)
   END_RUNG
   RUNG wire#w3
      Contact( #Use.Light )
      wire#w4
      I_Contact( #Alarm.H )
      I_Contact( #Alarm.L )
      Move(in := 1, out1 => #Status)
   END_RUNG
   RUNG wire#w4
      Contact( #Alarm.H )
      wire#w5
      Move(in := 3, out1 => #Status)
   END_RUNG
   RUNG wire#w4
      Contact( #Alarm.L )
   END_RUNG wire#w5
   RUNG wire#w2
      Contact( #Alarm.HH )
      wire#w6
      Move(in := 2, out1 => #Status)
   END_RUNG
   RUNG wire#w2
      Contact( #Alarm.LL )
   END_RUNG wire#w6
   RUNG wire#w2
      Contact( #Alarm.ST )
   END_RUNG wire#w6
   // the same network as SCL:
   IF NOT #Use.Status AND NOT #CMD.Hand THEN #Status := 0; END_IF;
   IF NOT #Use.Status AND #CMD.Hand THEN #Status := 7; END_IF;
   #_w1 := #Use.Status AND NOT #Alarm.HH AND NOT #Alarm.LL AND NOT #Alarm.ST;
   IF #_w1 AND NOT #Use.Light THEN #Status := 0; END_IF;
   #_w2 := #_w1 AND #Use.Light;
   IF #_w2 AND NOT #Alarm.H AND NOT #Alarm.L THEN #Status := 1; END_IF;
   IF #_w2 AND (#Alarm.H OR #Alarm.L) THEN #Status := 3; END_IF;
   IF #Use.Status AND (#Alarm.HH OR #Alarm.LL OR #Alarm.ST) THEN #Status := 2; END_IF;
END_REGION

REGION Network 26: Метка времени
   RUNG wire#powerrail
      Move(in := "Time_SYS_DB".RD_Time, out1 => #Time_DTL)
   END_RUNG
   // the same network as SCL:
   #Time_DTL := "Time_SYS_DB".RD_Time;
END_REGION
END_FUNCTION_BLOCK

FUNCTION "drv_Mode" : Void   // FC150, LAD
{ S7_Optimized_Access := 'FALSE' }
VERSION : 0.1
// stored: AutoNumber false, IsIECCheckEnabled false, SetENOAutomatically false, UDAEnableTagReadback false
   VAR_INPUT
      CMD : "CMD";   // Основные команды / Блок команд
      All_Block : Bool;   // Аварийная блокировка
   END_VAR
   VAR_OUTPUT
      Mode : Int;   // Режим работы
   END_VAR
BEGIN

REGION Network 1: Автоматический режим
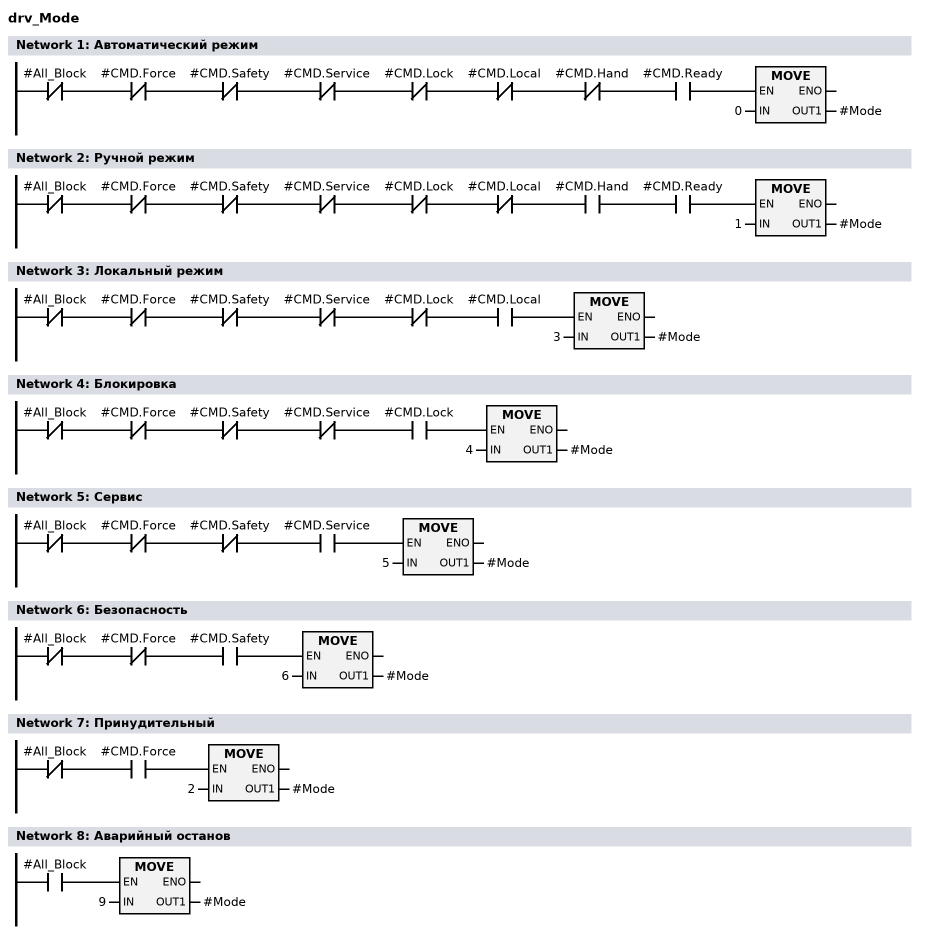
   RUNG wire#powerrail
      I_Contact( #All_Block )
      I_Contact( #CMD.Force )
      I_Contact( #CMD.Safety )
      I_Contact( #CMD.Service )
      I_Contact( #CMD.Lock )
      I_Contact( #CMD.Local )
      I_Contact( #CMD.Hand )
      Contact( #CMD.Ready )
      { S7_GenerateENO := "TRUE" } Move(in := 0, out1 => #Mode)
   END_RUNG
   // the same network as SCL:
   IF NOT #All_Block AND NOT #CMD.Force AND NOT #CMD.Safety AND NOT #CMD.Service AND NOT #CMD.Lock AND NOT #CMD.Local AND NOT #CMD.Hand AND #CMD.Ready THEN
       #Mode := 0;
   END_IF;
END_REGION

REGION Network 2: Ручной режим
   RUNG wire#powerrail
      I_Contact( #All_Block )
      I_Contact( #CMD.Force )
      I_Contact( #CMD.Safety )
      I_Contact( #CMD.Service )
      I_Contact( #CMD.Lock )
      I_Contact( #CMD.Local )
      Contact( #CMD.Hand )
      Contact( #CMD.Ready )
      { S7_GenerateENO := "TRUE" } Move(in := 1, out1 => #Mode)
   END_RUNG
   // the same network as SCL:
   IF NOT #All_Block AND NOT #CMD.Force AND NOT #CMD.Safety AND NOT #CMD.Service AND NOT #CMD.Lock AND NOT #CMD.Local AND #CMD.Hand AND #CMD.Ready THEN
       #Mode := 1;
   END_IF;
END_REGION

REGION Network 3: Локальный режим
   RUNG wire#powerrail
      I_Contact( #All_Block )
      I_Contact( #CMD.Force )
      I_Contact( #CMD.Safety )
      I_Contact( #CMD.Service )
      I_Contact( #CMD.Lock )
      Contact( #CMD.Local )
      { S7_GenerateENO := "TRUE" } Move(in := 3, out1 => #Mode)
   END_RUNG
   // the same network as SCL:
   IF NOT #All_Block AND NOT #CMD.Force AND NOT #CMD.Safety AND NOT #CMD.Service AND NOT #CMD.Lock AND #CMD.Local THEN
       #Mode := 3;
   END_IF;
END_REGION

REGION Network 4: Блокировка
   RUNG wire#powerrail
      I_Contact( #All_Block )
      I_Contact( #CMD.Force )
      I_Contact( #CMD.Safety )
      I_Contact( #CMD.Service )
      Contact( #CMD.Lock )
      { S7_GenerateENO := "TRUE" } Move(in := 4, out1 => #Mode)
   END_RUNG
   // the same network as SCL:
   IF NOT #All_Block AND NOT #CMD.Force AND NOT #CMD.Safety AND NOT #CMD.Service AND #CMD.Lock THEN
       #Mode := 4;
   END_IF;
END_REGION

REGION Network 5: Сервис
   RUNG wire#powerrail
      I_Contact( #All_Block )
      I_Contact( #CMD.Force )
      I_Contact( #CMD.Safety )
      Contact( #CMD.Service )
      { S7_GenerateENO := "TRUE" } Move(in := 5, out1 => #Mode)
   END_RUNG
   // the same network as SCL:
   IF NOT #All_Block AND NOT #CMD.Force AND NOT #CMD.Safety AND #CMD.Service THEN #Mode := 5; END_IF;
END_REGION

REGION Network 6: Безопасность
   RUNG wire#powerrail
      I_Contact( #All_Block )
      I_Contact( #CMD.Force )
      Contact( #CMD.Safety )
      { S7_GenerateENO := "TRUE" } Move(in := 6, out1 => #Mode)
   END_RUNG
   // the same network as SCL:
   IF NOT #All_Block AND NOT #CMD.Force AND #CMD.Safety THEN #Mode := 6; END_IF;
END_REGION

REGION Network 7: Принудительный
   RUNG wire#powerrail
      I_Contact( #All_Block )
      Contact( #CMD.Force )
      { S7_GenerateENO := "TRUE" } Move(in := 2, out1 => #Mode)
   END_RUNG
   // the same network as SCL:
   IF NOT #All_Block AND #CMD.Force THEN #Mode := 2; END_IF;
END_REGION

REGION Network 8: Аварийный останов
   RUNG wire#powerrail
      Contact( #All_Block )
      { S7_GenerateENO := "TRUE" } Move(in := 9, out1 => #Mode)
   END_RUNG
   // the same network as SCL:
   IF #All_Block THEN #Mode := 9; END_IF;
END_REGION
END_FUNCTION

FUNCTION_BLOCK "Time_R"   // FB91, LAD
{ S7_Optimized_Access := 'FALSE' }
VERSION : 0.1
// stored: AutoNumber false, IsIECCheckEnabled false, SetENOAutomatically false, UDAEnableTagReadback false
   VAR DB_SPECIFIC
      SP { S7_SetPoint := 'True'} : Real := 1.0;   // Уставка
      Now : Real;   // Текущий счёт
      One { S7_SetPoint := 'True'} : Real := 0.1;   // Вес импульса
      Progress : Real;   // Прогресс выполнения
      Start : Bool;   // Запуск
      "Exit" : Bool;   // Счёт завершён
      Pause : Bool;   // Пауза
      Reset : Bool;   // Сброс счёта
   END_VAR
   VAR_TEMP   // added for the SCL form of the ladder/FBD networks
      _w1 : Bool;
   END_VAR
BEGIN

REGION Network 1: Подсчёт времени
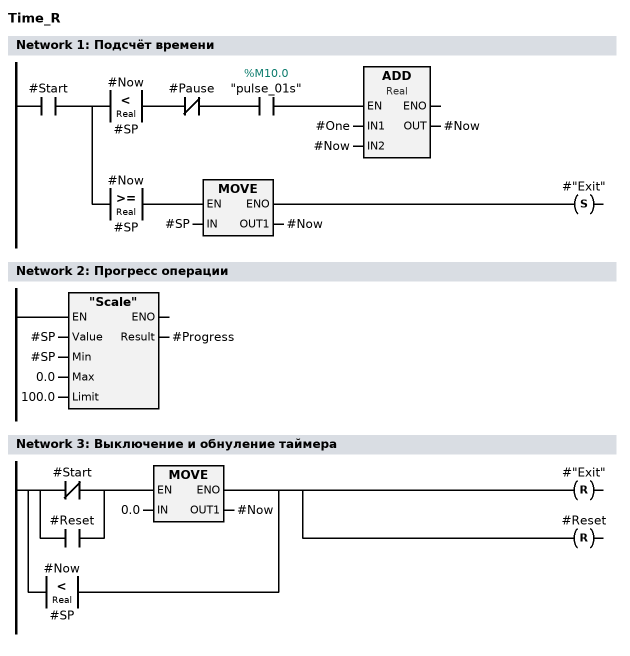
   RUNG wire#powerrail
      Contact( #Start )
      wire#w1
      { S7_Templates := "SrcType := Real" } LT_Contact(in1 := #Now, in2 := #SP)
      I_Contact( #Pause )
      Contact( "pulse_01s" )
      { S7_Templates := "SrcType := Real"; S7_GenerateENO := "TRUE" } Add(in1 := #One, in2 := #Now, out => #Now)
   END_RUNG
   RUNG wire#w1
      { S7_Templates := "SrcType := Real" } GE_Contact(in1 := #Now, in2 := #SP)
      Move(in := #SP, out1 => #Now)
      S_Coil( #"Exit" )
   END_RUNG
   // the same network as SCL:
   IF #Start AND (#Now < #SP) AND NOT #Pause AND "pulse_01s" THEN #Now := #One + #Now; END_IF;
   #_w1 := #Start AND (#Now >= #SP);
   IF #_w1 THEN
       #Now := #SP;
       #"Exit" := TRUE;
   END_IF;
END_REGION

REGION Network 2: Прогресс операции
   RUNG wire#powerrail
      "Scale"(Value := #SP, Min := #SP, Max := 0.0, Limit := 100.0, Result => #Progress)
   END_RUNG
   // the same network as SCL:
   "Scale"(Value := #SP, Min := #SP, Max := 0.0, Limit := 100.0, Result => #Progress);
END_REGION

REGION Network 3: Выключение и обнуление таймера
   RUNG wire#powerrail
      I_Contact( #Start )
      wire#w1
      { S7_GenerateENO := "TRUE" } Move(in := 0.0, out1 => #Now)
      wire#w2
      R_Coil( #"Exit" )
   END_RUNG
   RUNG wire#powerrail
      Contact( #Reset )
   END_RUNG wire#w1
   RUNG wire#powerrail
      { S7_Templates := "SrcType := Real" } LT_Contact(in1 := #Now, in2 := #SP)
   END_RUNG wire#w2
   RUNG wire#w2
      R_Coil( #Reset )
   END_RUNG
   // the same network as SCL:
   // ENO of a box is taken as its EN; it also drops when the box reports an error
   #_w1 := NOT #Start OR #Reset;
   IF #_w1 THEN #Now := 0.0; END_IF;
   IF #_w1 OR (#Now < #SP) THEN
       #"Exit" := FALSE;
       #Reset := FALSE;
   END_IF;
END_REGION
END_FUNCTION_BLOCK

FUNCTION_BLOCK "Gaz_status"
{ S7_Optimized_Access := 'FALSE' }
VERSION : 0.1
   VAR 
      Alarm : Word;
      H2_1_status : Int;
      H2_2_status : Int;
      Cl2_1_status : Int;
      Cl2_2_status : Int;
   END_VAR


BEGIN
	//датчик водорода 1
	IF NOT "DIx_1_DB".Gas_Chanel_1_1.Signal AND NOT "DIx_1_DB".Gas_Chanel_1_2.Signal THEN
	    #H2_1_status := 0;
	END_IF;
	IF "DIx_1_DB".Gas_Chanel_1_1.Signal OR "DIx_1_DB".Gas_Chanel_1_2.Signal THEN
	    #H2_1_status := 1;
	END_IF;
	IF "DIx_1_DB".Gas_Chanel_1_1.Signal AND "DIx_1_DB".Gas_Chanel_1_2.Signal THEN
	    #H2_1_status := 2;
	    #Alarm.%X0 := TRUE;
	END_IF;
	
	//датчик водорода 2
	IF NOT "DIx_1_DB".Gas_Chanel_2_1.Signal AND NOT "DIx_1_DB".Gas_Chanel_2_2.Signal THEN
	    #H2_2_status := 0;
	END_IF;
	IF "DIx_1_DB".Gas_Chanel_2_1.Signal OR "DIx_1_DB".Gas_Chanel_2_2.Signal THEN
	    #H2_2_status := 1;
	END_IF;
	IF "DIx_1_DB".Gas_Chanel_2_1.Signal AND "DIx_1_DB".Gas_Chanel_2_2.Signal THEN
	    #H2_2_status := 2;
	    #Alarm.%X1 := TRUE;
	END_IF;
	
	//датчик хлора 1
	IF NOT "DIx_1_DB".signal_11.Signal AND NOT "DIx_1_DB".signal_12.Signal THEN
	    #Cl2_1_status := 0;
	END_IF;
	IF "DIx_1_DB".signal_11.Signal OR "DIx_1_DB".signal_12.Signal THEN
	    #Cl2_1_status := 1;
	END_IF;
	IF "DIx_1_DB".signal_11.Signal AND "DIx_1_DB".signal_12.Signal THEN
	    #Cl2_1_status := 2;
	    #Alarm.%X2 := TRUE;
	END_IF;
	
	//датчик хлора 2
	IF NOT "DIx_1_DB".signal_10.Signal AND NOT "DIx_1_DB".signal_13.Signal THEN
	    #Cl2_2_status := 0;
	END_IF;
	IF "DIx_1_DB".signal_10.Signal OR "DIx_1_DB".signal_13.Signal THEN
	    #Cl2_2_status := 1;
	END_IF;
	IF "DIx_1_DB".signal_10.Signal AND "DIx_1_DB".signal_13.Signal THEN
	    #Cl2_2_status := 2;
	    #Alarm.%X3 := TRUE;
	END_IF;
	
	IF "Reset_All" THEN
	    #Alarm := 0;
	END_IF;
END_FUNCTION_BLOCK

FUNCTION_BLOCK "ModBus_TCP"   // FB40, LAD
TITLE = Блок опроса ModBus TCP
{ S7_Optimized_Access := 'FALSE' }
VERSION : 0.1
// ВНИМАНИЕ!  Через один аппаратный порт контроллера можно проводить множество различных опросов по ModBus TCP. Для этого у каждого экземпляра должен быть указан уникальный CONNECT.ID.
// 
// Для каждого уникального CONNECT.ID / внешней ветки / точки подключения (IP, RemotePort) рекомендуется использовать отдельный экземпляр функционального блока. Например, при использовании tGW-735 имеющего 3 порта подключения с RemotePort = 502, 503 и 504 соответственно (но общий IP адрес) рекомендуется использовать три отдельных блока ModBus_TCP с уникальными CONNECT.ID.
// 
// Каждая точка чтения/записи = 1 экземпляр DEV_Config, количество элементов в массиве можно менять по необходимости, итоговое количество элементов массива указывается в теге Limit.
// 
// Для режима чтения необходимо указать:
// - MODE = 0
// - Source_DB = 40 (номер DB Modbus_TCP_DB)
// - SourceOFFSET = 0
// - Target_DB = xx (номер DB, куда необходимо положить прочитанные данные)
// - Target_OFFSET = xx (номер байта, начиная с которого кладутся прочитанные данные в выбранный DB)
// 
// Для режима опроса необходимо указать:
// - MODE = 1
// - Source_DB = xx (номер DB, откуда необходимо взять данные для передачи)
// - Source_OFFSET = xx (номер байта, начиная с которого берутся данные для передачи)
// - Target_DB = 40 (номер DB Modbus_TCP_DB)
// - Target_OFFSET = 0
// stored: AutoNumber false, IsIECCheckEnabled false, SetENOAutomatically false, UDAEnableTagReadback false
   VAR DB_SPECIFIC
      COM_Control : Struct
         Enable { S7_SetPoint := 'True'} : Bool := true;   // Использовать коммуникацию
         Start : Bool;   // Начать опрос
         Reset : Bool;   // Сброс драйвера
         REQ_NDR : Bool;   // Опрос завершён
         REQ_DR : Bool;   // Опрос в процессе
         REQ_Error : Bool;   // Опрос - ошибка
         REQ_Status : Word;   // Опрос - код состояния
         Error_Code : Word;   // Опрос - код аварии
         Status : Int;   // 1 - успешно, 2 - нет ответа, 3 - ошибка параметров
      END_STRUCT;
      CONNECT { S7_SetPoint := 'True'} : TCON_IP_v4;
   END_VAR
   // CONNECT.InterfaceId := 64;
   // CONNECT.ID := 16#0001;
   // CONNECT.ConnectionType := 16#0B;
   // CONNECT.ActiveEstablished := TRUE;
   // CONNECT.RemoteAddress.ADDR[1..4] := 0;
   // CONNECT.RemotePort := 502;
   // CONNECT.LocalPort := 0;
BEGIN

REGION Network 1
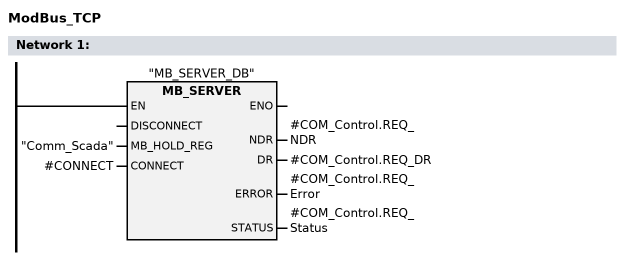
   RUNG wire#powerrail
      "MB_SERVER_DB".MB_SERVER(DISCONNECT :=, MB_HOLD_REG := "Comm_Scada", CONNECT := #CONNECT, NDR => #COM_Control.REQ_NDR, DR => #COM_Control.REQ_DR, ERROR => #COM_Control.REQ_Error, STATUS => #COM_Control.REQ_Status)
   END_RUNG
   // the same network as SCL:
   "MB_SERVER_DB"(MB_HOLD_REG := "Comm_Scada",   // MB_SERVER
                  CONNECT := #CONNECT,
                  NDR => #COM_Control.REQ_NDR,
                  DR => #COM_Control.REQ_DR,
                  ERROR => #COM_Control.REQ_Error,
                  STATUS => #COM_Control.REQ_Status);
END_REGION
END_FUNCTION_BLOCK

FUNCTION_BLOCK "Logick"   // FB1, LAD
{ S7_Optimized_Access := 'FALSE' }
VERSION : 0.1
// stored: AutoNumber true, IsIECCheckEnabled false, SetENOAutomatically false, UDAEnableTagReadback false
   VAR DB_SPECIFIC
      Start_ELZ : Bool;   // Запуск электролизеров (приготовления)
      REQ_Wash : Bool;   // Запрос запуска промывки
      Force_Wash : Bool;   // Принудительная промывка
      ELZ : Bool;
      Local : Bool;   // Дистанционное управление
      Step_Wash : Int;   // Шаг промывки
      ELZ_LED : Int;   // Подсветка электролизера на панели
      RM_1 { S7_SetPoint := 'True'} : Real;
      Alarm : Word;   // Слово аварий
      Alarms : Struct
         Gas : Bool;   // Остановка по загазованности
         ELZ_AHLS : Bool;   // Электролизер - переполнение поддона
      END_STRUCT;
   END_VAR
   VAR
      ELZ_1 { S7_SetPoint := 'True'} : "ELZ";
   END_VAR
   VAR DB_SPECIFIC
      Days : Struct   // Расписание промывки (дни)
         D_1 : Bool;   // Расписание промывки (день 1)
         D_2 : Bool;   // Расписание промывки (день 2)
         D_3 : Bool;   // Расписание промывки (день 3)
         D_4 : Bool;   // Расписание промывки (день 4)
         D_5 : Bool;   // Расписание промывки (день 5)
         D_6 : Bool;   // Расписание промывки (день 6)
         D_7 : Bool;   // Расписание промывки (день 7)
      END_STRUCT;
      Houres : Struct   // Расписание промывки (часы)
         H_D_1 : Int;   // Расписание промывки (часы 1 дня)
         H_D_2 : Int;   // Расписание промывки (часы 2 дня)
         H_D_3 : Int;   // Расписание промывки (часы 3 дня)
         H_D_4 : Int;   // Расписание промывки (часы 4 дня)
         H_D_5 : Int;   // Расписание промывки (часы 5 дня)
         H_D_6 : Int;   // Расписание промывки (часы 6 дня)
         H_D_7 : Int;   // Расписание промывки (часы 7 дня)
      END_STRUCT;
      Minutes : Struct   // Расписание промывки (минуты)
         M_D_1 : Int;   // Расписание промывки (минуты 1 дня)
         M_D_2 : Int;   // Расписание промывки (минуты 2 дня)
         M_D_3 : Int;   // Расписание промывки (минуты 3 дня)
         M_D_4 : Int;   // Расписание промывки (минуты 4 дня)
         M_D_5 : Int;   // Расписание промывки (минуты 5 дня)
         M_D_6 : Int;   // Расписание промывки (минуты 6 дня)
         M_D_7 : Int;   // Расписание промывки (минуты 7 дня)
      END_STRUCT;
   END_VAR
   VAR
      T_Wash { S7_SetPoint := 'True'} : "Time_M";   // Время промывки
   END_VAR
   VAR_TEMP   // added for the SCL form of the ladder/FBD networks
      _w1 : Bool;
      _w2 : Bool;
   END_VAR
BEGIN

REGION Network 1: Электролизеры
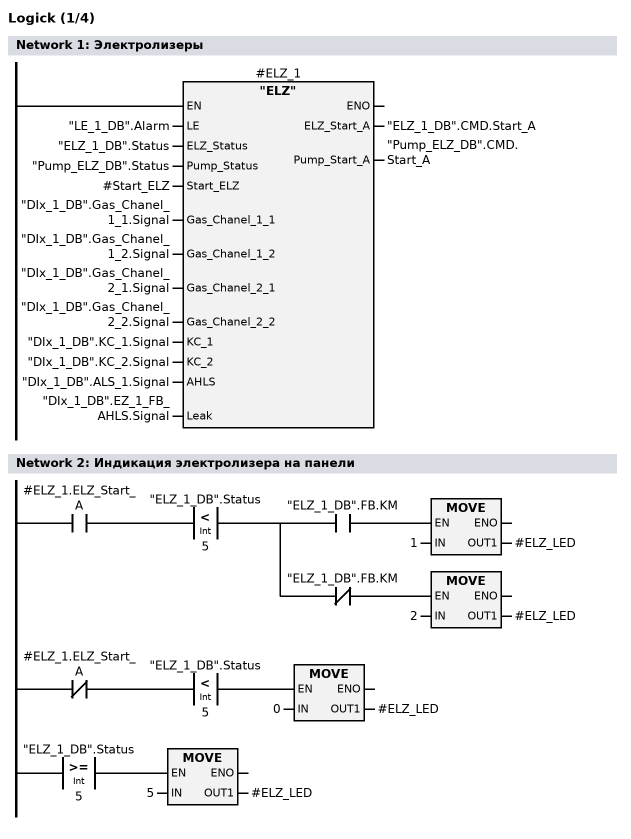
   RUNG wire#powerrail
      #ELZ_1(LE := "LE_1_DB".Alarm, ELZ_Status := "ELZ_1_DB".Status, Pump_Status := "Pump_ELZ_DB".Status, Start_ELZ := #Start_ELZ, Gas_Chanel_1_1 := "DIx_1_DB".Gas_Chanel_1_1.Signal, Gas_Chanel_1_2 := "DIx_1_DB".Gas_Chanel_1_2.Signal, Gas_Chanel_2_1 := "DIx_1_DB".Gas_Chanel_2_1.Signal, Gas_Chanel_2_2 := "DIx_1_DB".Gas_Chanel_2_2.Signal, KC_1 := "DIx_1_DB".KC_1.Signal, KC_2 := "DIx_1_DB".KC_2.Signal, AHLS := "DIx_1_DB".ALS_1.Signal, Leak := "DIx_1_DB".EZ_1_FB_AHLS.Signal, ELZ_Start_A => "ELZ_1_DB".CMD.Start_A, Pump_Start_A => "Pump_ELZ_DB".CMD.Start_A)
   END_RUNG
   // the same network as SCL:
   #ELZ_1(LE := "LE_1_DB".Alarm,   // "ELZ"
          ELZ_Status := "ELZ_1_DB".Status,
          Pump_Status := "Pump_ELZ_DB".Status,
          Start_ELZ := #Start_ELZ,
          Gas_Chanel_1_1 := "DIx_1_DB".Gas_Chanel_1_1.Signal,
          Gas_Chanel_1_2 := "DIx_1_DB".Gas_Chanel_1_2.Signal,
          Gas_Chanel_2_1 := "DIx_1_DB".Gas_Chanel_2_1.Signal,
          Gas_Chanel_2_2 := "DIx_1_DB".Gas_Chanel_2_2.Signal,
          KC_1 := "DIx_1_DB".KC_1.Signal,
          KC_2 := "DIx_1_DB".KC_2.Signal,
          AHLS := "DIx_1_DB".ALS_1.Signal,
          Leak := "DIx_1_DB".EZ_1_FB_AHLS.Signal,
          ELZ_Start_A => "ELZ_1_DB".CMD.Start_A,
          Pump_Start_A => "Pump_ELZ_DB".CMD.Start_A);
END_REGION

REGION Network 2: Индикация электролизера на панели
   RUNG wire#powerrail
      Contact( #ELZ_1.ELZ_Start_A )
      { S7_Templates := "SrcType := Int" } LT_Contact(in1 := "ELZ_1_DB".Status, in2 := 5)
      wire#w1
      Contact( "ELZ_1_DB".FB.KM )
      Move(in := 1, out1 => #ELZ_LED)
   END_RUNG
   RUNG wire#w1
      I_Contact( "ELZ_1_DB".FB.KM )
      Move(in := 2, out1 => #ELZ_LED)
   END_RUNG
   RUNG wire#powerrail
      I_Contact( #ELZ_1.ELZ_Start_A )
      { S7_Templates := "SrcType := Int" } LT_Contact(in1 := "ELZ_1_DB".Status, in2 := 5)
      Move(in := 0, out1 => #ELZ_LED)
   END_RUNG
   RUNG wire#powerrail
      { S7_Templates := "SrcType := Int" } GE_Contact(in1 := "ELZ_1_DB".Status, in2 := 5)
      Move(in := 5, out1 => #ELZ_LED)
   END_RUNG
   // the same network as SCL:
   #_w1 := #ELZ_1.ELZ_Start_A AND ("ELZ_1_DB".Status < 5);
   IF #_w1 AND "ELZ_1_DB".FB.KM THEN #ELZ_LED := 1; END_IF;
   IF #_w1 AND NOT "ELZ_1_DB".FB.KM THEN #ELZ_LED := 2; END_IF;
   IF NOT #ELZ_1.ELZ_Start_A AND ("ELZ_1_DB".Status < 5) THEN #ELZ_LED := 0; END_IF;
   IF "ELZ_1_DB".Status >= 5 THEN #ELZ_LED := 5; END_IF;
END_REGION

REGION Network 3: Запрос промывки фильтров (Пришло время в расписании)
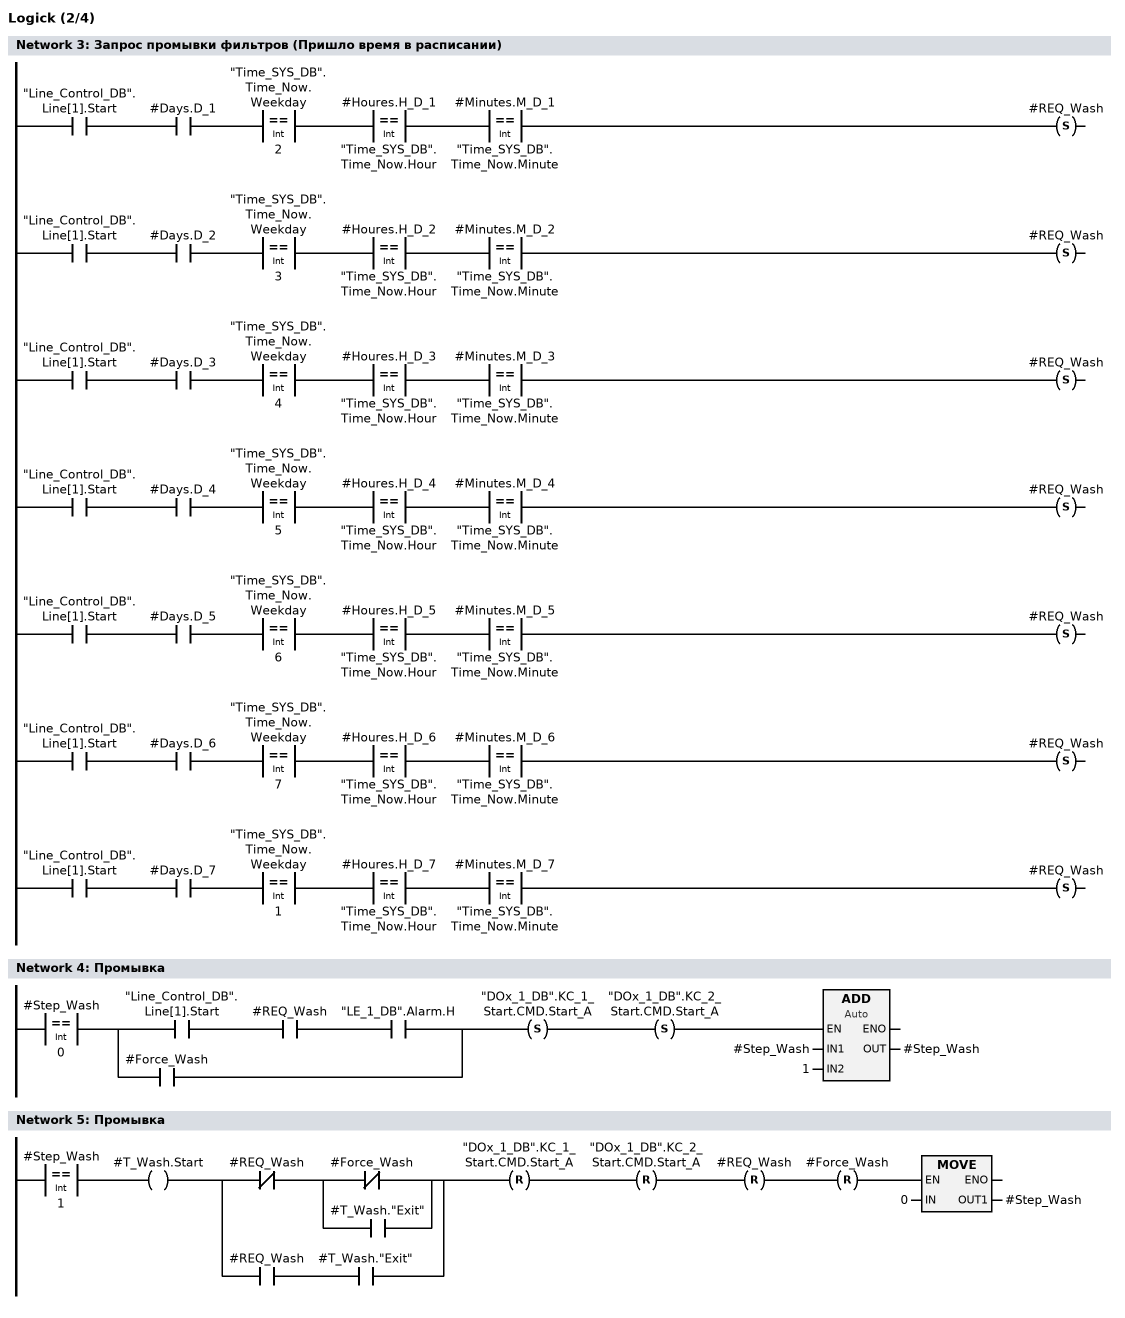
   RUNG wire#powerrail
      Contact( "Line_Control_DB".Line[1].Start )
      Contact( #Days.D_1 )
      { S7_Templates := "SrcType := Int" } EQ_Contact(in1 := "Time_SYS_DB".Time_Now.Weekday, in2 := 2)
      { S7_Templates := "SrcType := Int" } EQ_Contact(in1 := #Houres.H_D_1, in2 := "Time_SYS_DB".Time_Now.Hour)
      { S7_Templates := "SrcType := Int" } EQ_Contact(in1 := #Minutes.M_D_1, in2 := "Time_SYS_DB".Time_Now.Minute)
      S_Coil( #REQ_Wash )
   END_RUNG
   RUNG wire#powerrail
      Contact( "Line_Control_DB".Line[1].Start )
      Contact( #Days.D_2 )
      { S7_Templates := "SrcType := Int" } EQ_Contact(in1 := "Time_SYS_DB".Time_Now.Weekday, in2 := 3)
      { S7_Templates := "SrcType := Int" } EQ_Contact(in1 := #Houres.H_D_2, in2 := "Time_SYS_DB".Time_Now.Hour)
      { S7_Templates := "SrcType := Int" } EQ_Contact(in1 := #Minutes.M_D_2, in2 := "Time_SYS_DB".Time_Now.Minute)
      S_Coil( #REQ_Wash )
   END_RUNG
   RUNG wire#powerrail
      Contact( "Line_Control_DB".Line[1].Start )
      Contact( #Days.D_3 )
      { S7_Templates := "SrcType := Int" } EQ_Contact(in1 := "Time_SYS_DB".Time_Now.Weekday, in2 := 4)
      { S7_Templates := "SrcType := Int" } EQ_Contact(in1 := #Houres.H_D_3, in2 := "Time_SYS_DB".Time_Now.Hour)
      { S7_Templates := "SrcType := Int" } EQ_Contact(in1 := #Minutes.M_D_3, in2 := "Time_SYS_DB".Time_Now.Minute)
      S_Coil( #REQ_Wash )
   END_RUNG
   RUNG wire#powerrail
      Contact( "Line_Control_DB".Line[1].Start )
      Contact( #Days.D_4 )
      { S7_Templates := "SrcType := Int" } EQ_Contact(in1 := "Time_SYS_DB".Time_Now.Weekday, in2 := 5)
      { S7_Templates := "SrcType := Int" } EQ_Contact(in1 := #Houres.H_D_4, in2 := "Time_SYS_DB".Time_Now.Hour)
      { S7_Templates := "SrcType := Int" } EQ_Contact(in1 := #Minutes.M_D_4, in2 := "Time_SYS_DB".Time_Now.Minute)
      S_Coil( #REQ_Wash )
   END_RUNG
   RUNG wire#powerrail
      Contact( "Line_Control_DB".Line[1].Start )
      Contact( #Days.D_5 )
      { S7_Templates := "SrcType := Int" } EQ_Contact(in1 := "Time_SYS_DB".Time_Now.Weekday, in2 := 6)
      { S7_Templates := "SrcType := Int" } EQ_Contact(in1 := #Houres.H_D_5, in2 := "Time_SYS_DB".Time_Now.Hour)
      { S7_Templates := "SrcType := Int" } EQ_Contact(in1 := #Minutes.M_D_5, in2 := "Time_SYS_DB".Time_Now.Minute)
      S_Coil( #REQ_Wash )
   END_RUNG
   RUNG wire#powerrail
      Contact( "Line_Control_DB".Line[1].Start )
      Contact( #Days.D_6 )
      { S7_Templates := "SrcType := Int" } EQ_Contact(in1 := "Time_SYS_DB".Time_Now.Weekday, in2 := 7)
      { S7_Templates := "SrcType := Int" } EQ_Contact(in1 := #Houres.H_D_6, in2 := "Time_SYS_DB".Time_Now.Hour)
      { S7_Templates := "SrcType := Int" } EQ_Contact(in1 := #Minutes.M_D_6, in2 := "Time_SYS_DB".Time_Now.Minute)
      S_Coil( #REQ_Wash )
   END_RUNG
   RUNG wire#powerrail
      Contact( "Line_Control_DB".Line[1].Start )
      Contact( #Days.D_7 )
      { S7_Templates := "SrcType := Int" } EQ_Contact(in1 := "Time_SYS_DB".Time_Now.Weekday, in2 := 1)
      { S7_Templates := "SrcType := Int" } EQ_Contact(in1 := #Houres.H_D_7, in2 := "Time_SYS_DB".Time_Now.Hour)
      { S7_Templates := "SrcType := Int" } EQ_Contact(in1 := #Minutes.M_D_7, in2 := "Time_SYS_DB".Time_Now.Minute)
      S_Coil( #REQ_Wash )
   END_RUNG
   // the same network as SCL:
   IF "Line_Control_DB".Line[1].Start AND #Days.D_1 AND ("Time_SYS_DB".Time_Now.Weekday = 2) AND (#Houres.H_D_1 = "Time_SYS_DB".Time_Now.Hour) AND (#Minutes.M_D_1 = "Time_SYS_DB".Time_Now.Minute) THEN
       #REQ_Wash := TRUE;
   END_IF;
   IF "Line_Control_DB".Line[1].Start AND #Days.D_2 AND ("Time_SYS_DB".Time_Now.Weekday = 3) AND (#Houres.H_D_2 = "Time_SYS_DB".Time_Now.Hour) AND (#Minutes.M_D_2 = "Time_SYS_DB".Time_Now.Minute) THEN
       #REQ_Wash := TRUE;
   END_IF;
   IF "Line_Control_DB".Line[1].Start AND #Days.D_3 AND ("Time_SYS_DB".Time_Now.Weekday = 4) AND (#Houres.H_D_3 = "Time_SYS_DB".Time_Now.Hour) AND (#Minutes.M_D_3 = "Time_SYS_DB".Time_Now.Minute) THEN
       #REQ_Wash := TRUE;
   END_IF;
   IF "Line_Control_DB".Line[1].Start AND #Days.D_4 AND ("Time_SYS_DB".Time_Now.Weekday = 5) AND (#Houres.H_D_4 = "Time_SYS_DB".Time_Now.Hour) AND (#Minutes.M_D_4 = "Time_SYS_DB".Time_Now.Minute) THEN
       #REQ_Wash := TRUE;
   END_IF;
   IF "Line_Control_DB".Line[1].Start AND #Days.D_5 AND ("Time_SYS_DB".Time_Now.Weekday = 6) AND (#Houres.H_D_5 = "Time_SYS_DB".Time_Now.Hour) AND (#Minutes.M_D_5 = "Time_SYS_DB".Time_Now.Minute) THEN
       #REQ_Wash := TRUE;
   END_IF;
   IF "Line_Control_DB".Line[1].Start AND #Days.D_6 AND ("Time_SYS_DB".Time_Now.Weekday = 7) AND (#Houres.H_D_6 = "Time_SYS_DB".Time_Now.Hour) AND (#Minutes.M_D_6 = "Time_SYS_DB".Time_Now.Minute) THEN
       #REQ_Wash := TRUE;
   END_IF;
   IF "Line_Control_DB".Line[1].Start AND #Days.D_7 AND ("Time_SYS_DB".Time_Now.Weekday = 1) AND (#Houres.H_D_7 = "Time_SYS_DB".Time_Now.Hour) AND (#Minutes.M_D_7 = "Time_SYS_DB".Time_Now.Minute) THEN
       #REQ_Wash := TRUE;
   END_IF;
END_REGION

REGION Network 4: Промывка
   RUNG wire#powerrail
      { S7_Templates := "SrcType := Int" } EQ_Contact(in1 := #Step_Wash, in2 := 0)
      wire#w1
      Contact( "Line_Control_DB".Line[1].Start )
      Contact( #REQ_Wash )
      Contact( "LE_1_DB".Alarm.H )
      wire#w2
      S_Coil( "DOx_1_DB".KC_1_Start.CMD.Start_A )
      S_Coil( "DOx_1_DB".KC_2_Start.CMD.Start_A )
      Add(in1 := #Step_Wash, in2 := 1, out => #Step_Wash)
   END_RUNG
   RUNG wire#w1
      Contact( #Force_Wash )
   END_RUNG wire#w2
   // the same network as SCL:
   IF (#Step_Wash = 0) AND (("Line_Control_DB".Line[1].Start AND #REQ_Wash AND "LE_1_DB".Alarm.H) OR #Force_Wash) THEN
       "DOx_1_DB".KC_1_Start.CMD.Start_A := TRUE;
       "DOx_1_DB".KC_2_Start.CMD.Start_A := TRUE;
       #Step_Wash := #Step_Wash + 1;
   END_IF;
END_REGION

REGION Network 5: Промывка
   RUNG wire#powerrail
      { S7_Templates := "SrcType := Int" } EQ_Contact(in1 := #Step_Wash, in2 := 1)
      Coil( #T_Wash.Start )
      wire#w1
      I_Contact( #REQ_Wash )
      wire#w2
      I_Contact( #Force_Wash )
      wire#w3
      R_Coil( "DOx_1_DB".KC_1_Start.CMD.Start_A )
      R_Coil( "DOx_1_DB".KC_2_Start.CMD.Start_A )
      R_Coil( #REQ_Wash )
      R_Coil( #Force_Wash )
      Move(in := 0, out1 => #Step_Wash)
   END_RUNG
   RUNG wire#w2
      Contact( #T_Wash."Exit" )
   END_RUNG wire#w3
   RUNG wire#w1
      Contact( #REQ_Wash )
      Contact( #T_Wash."Exit" )
   END_RUNG wire#w3
   // the same network as SCL:
   #T_Wash.Start := #Step_Wash = 1;
   IF #T_Wash.Start AND ((NOT #REQ_Wash AND (NOT #Force_Wash OR #T_Wash."Exit")) OR (#REQ_Wash AND #T_Wash."Exit")) THEN
       "DOx_1_DB".KC_1_Start.CMD.Start_A := FALSE;
       "DOx_1_DB".KC_2_Start.CMD.Start_A := FALSE;
   END_IF;
   #_w1 := #T_Wash.Start AND ((NOT #REQ_Wash AND (NOT #Force_Wash OR #T_Wash."Exit")) OR (#REQ_Wash AND #T_Wash."Exit"));
   IF #_w1 THEN
       #REQ_Wash := FALSE;
       #Force_Wash := FALSE;
       #Step_Wash := 0;
   END_IF;
END_REGION

REGION Network 6: Блокировка и авария насосов 1 и 2 по низкому уровню и неисправности датчиков
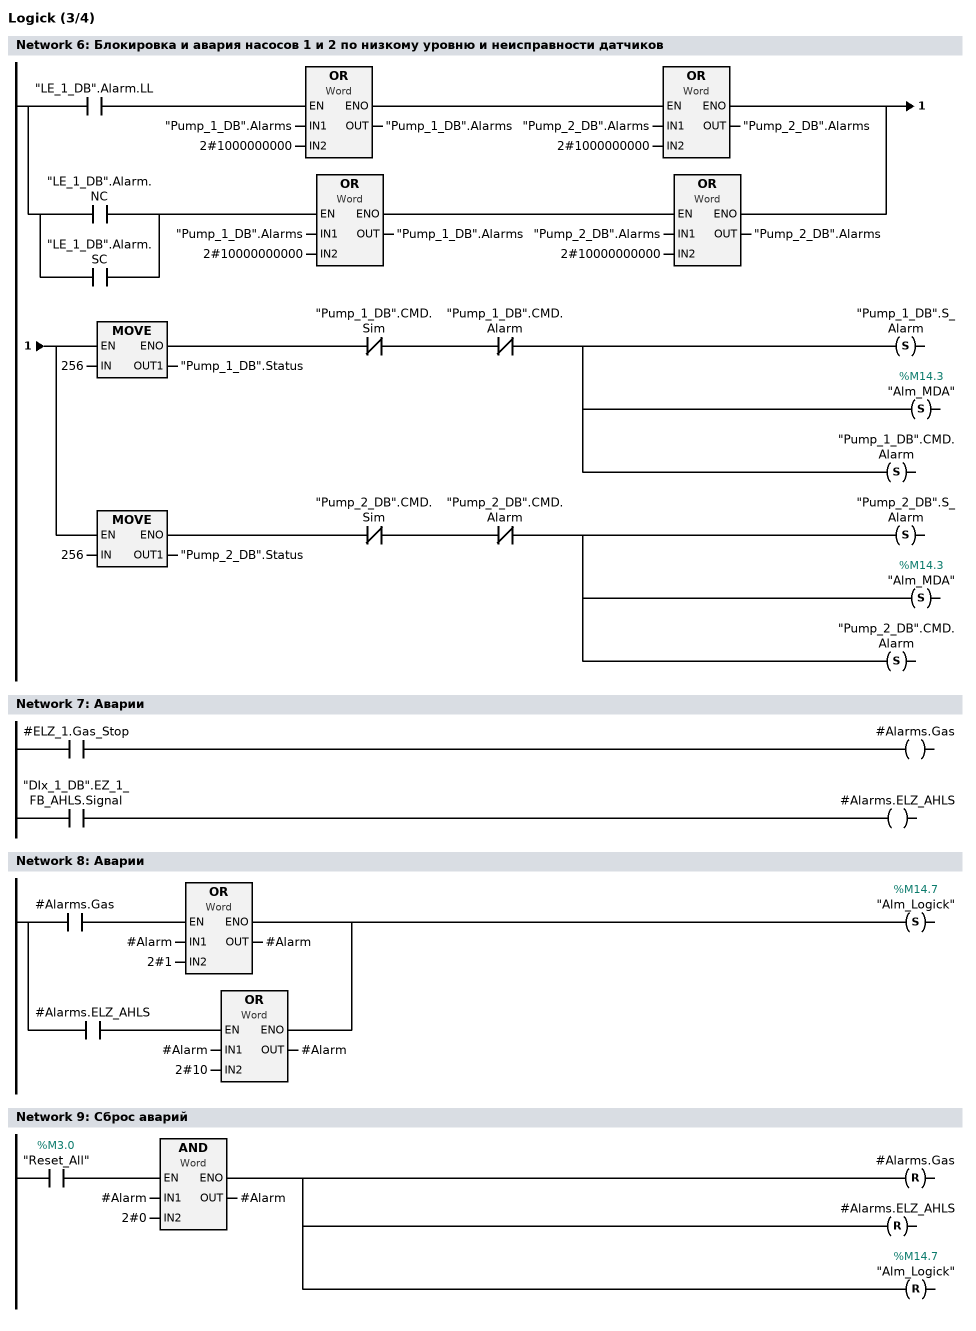
   // ENO of a box is taken as its EN; it also drops when the box reports an error
   IF "LE_1_DB".Alarm.LL THEN
       "Pump_1_DB".Alarms := "Pump_1_DB".Alarms OR 2#1000000000;
       "Pump_2_DB".Alarms := "Pump_2_DB".Alarms OR 2#1000000000;
   END_IF;
   #_w1 := "LE_1_DB".Alarm.NC OR "LE_1_DB".Alarm.SC;
   IF #_w1 THEN
       "Pump_1_DB".Alarms := "Pump_1_DB".Alarms OR 2#10000000000;
       "Pump_2_DB".Alarms := "Pump_2_DB".Alarms OR 2#10000000000;
   END_IF;
   #_w2 := "LE_1_DB".Alarm.LL OR #_w1;
   IF #_w2 THEN "Pump_1_DB".Status := 256; END_IF;
   IF #_w2 AND NOT "Pump_1_DB".CMD.Sim AND NOT "Pump_1_DB".CMD.Alarm THEN
       "Pump_1_DB".S_Alarm := TRUE;
       "Alm_MDA" := TRUE;
       "Pump_1_DB".CMD.Alarm := TRUE;
   END_IF;
   IF #_w2 THEN "Pump_2_DB".Status := 256; END_IF;
   IF #_w2 AND NOT "Pump_2_DB".CMD.Sim AND NOT "Pump_2_DB".CMD.Alarm THEN
       "Pump_2_DB".S_Alarm := TRUE;
       "Alm_MDA" := TRUE;
       "Pump_2_DB".CMD.Alarm := TRUE;
   END_IF;
END_REGION

REGION Network 7: Аварии
   RUNG wire#powerrail
      Contact( #ELZ_1.Gas_Stop )
      Coil( #Alarms.Gas )
   END_RUNG
   RUNG wire#powerrail
      Contact( "DIx_1_DB".EZ_1_FB_AHLS.Signal )
      Coil( #Alarms.ELZ_AHLS )
   END_RUNG
   // the same network as SCL:
   #Alarms.Gas := #ELZ_1.Gas_Stop;
   #Alarms.ELZ_AHLS := "DIx_1_DB".EZ_1_FB_AHLS.Signal;
END_REGION

REGION Network 8: Аварии
   IF #Alarms.Gas THEN #Alarm := #Alarm OR 2#1; END_IF;
   IF #Alarms.ELZ_AHLS THEN #Alarm := #Alarm OR 2#10; END_IF;
   IF #Alarms.Gas OR #Alarms.ELZ_AHLS THEN "Alm_Logick" := TRUE; END_IF;
END_REGION

REGION Network 9: Сброс аварий
   RUNG wire#powerrail
      Contact( "Reset_All" )
      { S7_Templates := "SrcType := Word"; S7_GenerateENO := "TRUE" } And(in1 := #Alarm, in2 := 2#0, out => #Alarm)
      wire#w1
      R_Coil( #Alarms.Gas )
   END_RUNG
   RUNG wire#w1
      R_Coil( #Alarms.ELZ_AHLS )
   END_RUNG
   RUNG wire#w1
      R_Coil( "Alm_Logick" )
   END_RUNG
   // the same network as SCL:
   IF "Reset_All" THEN
       #Alarm := #Alarm AND 2#0;
       #Alarms.Gas := FALSE;
       #Alarms.ELZ_AHLS := FALSE;
       "Alm_Logick" := FALSE;
   END_IF;
END_REGION

REGION Network 10: Сигнальная колонна
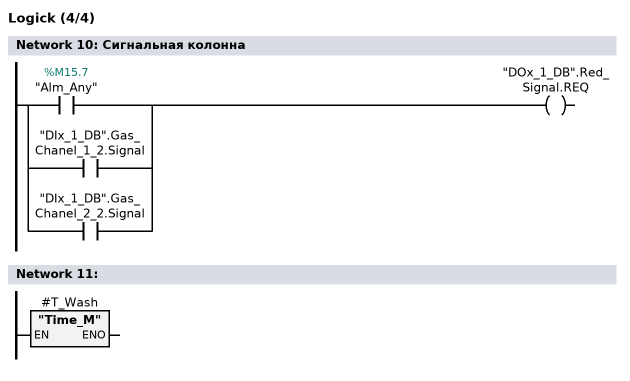
   RUNG wire#powerrail
      Contact( "Alm_Any" )
      wire#w1
      Coil( "DOx_1_DB".Red_Signal.REQ )
   END_RUNG
   RUNG wire#powerrail
      Contact( "DIx_1_DB".Gas_Chanel_1_2.Signal )
   END_RUNG wire#w1
   RUNG wire#powerrail
      Contact( "DIx_1_DB".Gas_Chanel_2_2.Signal )
   END_RUNG wire#w1
   // the same network as SCL:
   "DOx_1_DB".Red_Signal.REQ := "Alm_Any" OR "DIx_1_DB".Gas_Chanel_1_2.Signal OR "DIx_1_DB".Gas_Chanel_2_2.Signal;
END_REGION

REGION Network 11
   RUNG wire#powerrail
      #T_Wash()
   END_RUNG
   // the same network as SCL:
   #T_Wash();   // "Time_M"
END_REGION
END_FUNCTION_BLOCK

FUNCTION_BLOCK "ELZ"   // FB3, LAD
{ S7_Optimized_Access := 'FALSE' }
VERSION : 0.1
// stored: AutoNumber true, IsIECCheckEnabled false, SetENOAutomatically false, UDAEnableTagReadback false
   VAR_INPUT
      LE : Struct   // Границы датчика
         ST : Bool;   // Общая неисправность
         HH : Bool;   // сработала авария по аварийно высокму уровню
         H : Bool;   // сработало предупреждение по высокому уровню
         L : Bool;   // сработало предупреждение по низкому уровню
         LL : Bool;   // сработало предупрждение по аварийно низкому уровню
         NC : Bool;   // обрыв линии
         SC : Bool;   // короткое замыкание
      END_STRUCT;
      ELZ_Status : Int;   // Статус электролизера
      Pump_Status : Int;   // Статус насоса
      Start_ELZ : Bool;   // Старт электролизера
      Gas_Chanel_1_1 : Bool;   // Датчик загазованности
      Gas_Chanel_1_2 : Bool;   // Датчик загазованности
      Gas_Chanel_2_1 : Bool;   // Датчик загазованности
      Gas_Chanel_2_2 : Bool;   // Датчик загазованности
      KC_1 : Bool;   // Промывочные клапана с фильтров
      KC_2 : Bool;   // Промывочные клапана с фильтров
      AHLS : Bool;   // Верхний аварийный датчик уровня
      Leak : Bool;   // Переполнение поддона
   END_VAR
   VAR_OUTPUT
      ELZ_Start_A : Bool;   // Запуск электролизера
      Pump_Start_A : Bool;   // Запуск насоса
   END_VAR
   VAR DB_SPECIFIC
      Mode : Bool;   // 0 - предупреждение, 1 - остановка через таймер
      Wash : Bool;   // Идет промывка (для панели)
      Gas_Stop : Bool;   // Запрет запуска при загазованности
      Gas : Int;   // Предупреждение о загазованности на панели
      "Step" : Int;
   END_VAR
   VAR
      T_Gas { S7_SetPoint := 'True'} : "Time_M";
      T_ELZ_Start { S7_SetPoint := 'True'} : "Time_M";   // Задержка запуска электролизера
   END_VAR
   // T_ELZ_Start.SP_S := 10;
   VAR_TEMP   // added for the SCL form of the ladder/FBD networks
      _w1 : Bool;
   END_VAR
BEGIN

REGION Network 1: Старт / Выключение электролизера по высокому уровню в баке и по загазованности (порог 2)
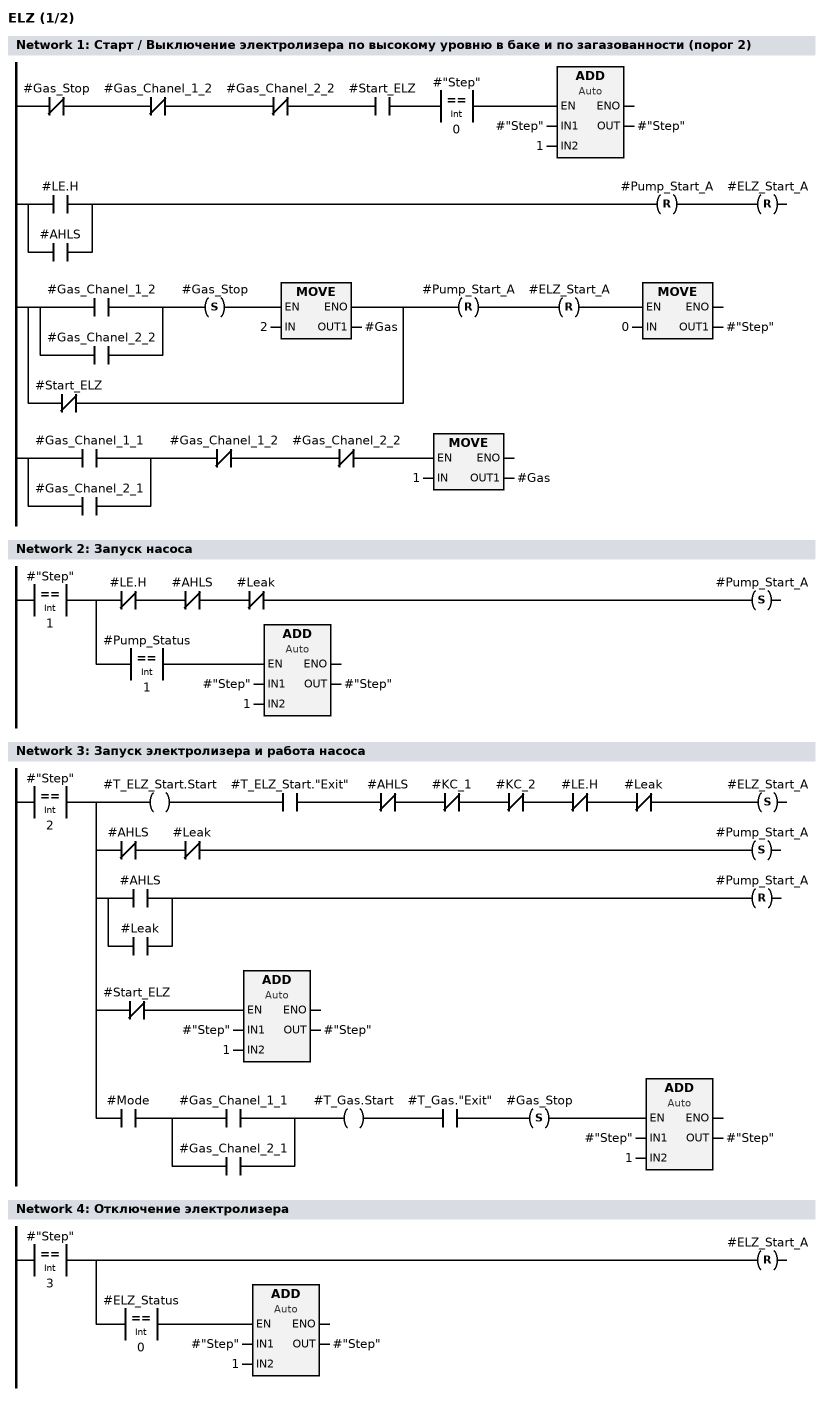
   RUNG wire#powerrail
      I_Contact( #Gas_Stop )
      I_Contact( #Gas_Chanel_1_2 )
      I_Contact( #Gas_Chanel_2_2 )
      Contact( #Start_ELZ )
      { S7_Templates := "SrcType := Int" } EQ_Contact(in1 := #"Step", in2 := 0)
      Add(in1 := #"Step", in2 := 1, out => #"Step")
   END_RUNG
   RUNG wire#powerrail
      Contact( #LE.H )
      wire#w1
      R_Coil( #Pump_Start_A )
      R_Coil( #ELZ_Start_A )
   END_RUNG
   RUNG wire#powerrail
      Contact( #AHLS )
   END_RUNG wire#w1
   RUNG wire#powerrail
      Contact( #Gas_Chanel_1_2 )
      wire#w2
      S_Coil( #Gas_Stop )
      Move(in := 2, out1 => #Gas)
      wire#w3
      R_Coil( #Pump_Start_A )
      R_Coil( #ELZ_Start_A )
      Move(in := 0, out1 => #"Step")
   END_RUNG
   RUNG wire#powerrail
      Contact( #Gas_Chanel_2_2 )
   END_RUNG wire#w2
   RUNG wire#powerrail
      I_Contact( #Start_ELZ )
   END_RUNG wire#w3
   RUNG wire#powerrail
      Contact( #Gas_Chanel_1_1 )
      wire#w4
      I_Contact( #Gas_Chanel_1_2 )
      I_Contact( #Gas_Chanel_2_2 )
      Move(in := 1, out1 => #Gas)
   END_RUNG
   RUNG wire#powerrail
      Contact( #Gas_Chanel_2_1 )
   END_RUNG wire#w4
   // the same network as SCL:
   IF NOT #Gas_Stop AND NOT #Gas_Chanel_1_2 AND NOT #Gas_Chanel_2_2 AND #Start_ELZ AND (#"Step" = 0) THEN
       #"Step" := #"Step" + 1;
   END_IF;
   IF #LE.H OR #AHLS THEN
       #Pump_Start_A := FALSE;
       #ELZ_Start_A := FALSE;
   END_IF;
   #_w1 := #Gas_Chanel_1_2 OR #Gas_Chanel_2_2;
   IF #_w1 THEN
       #Gas_Stop := TRUE;
       #Gas := 2;
   END_IF;
   IF #_w1 OR NOT #Start_ELZ THEN
       #Pump_Start_A := FALSE;
       #ELZ_Start_A := FALSE;
       #"Step" := 0;
   END_IF;
   IF (#Gas_Chanel_1_1 OR #Gas_Chanel_2_1) AND NOT #Gas_Chanel_1_2 AND NOT #Gas_Chanel_2_2 THEN
       #Gas := 1;
   END_IF;
END_REGION

REGION Network 2: Запуск насоса
   RUNG wire#powerrail
      { S7_Templates := "SrcType := Int" } EQ_Contact(in1 := #"Step", in2 := 1)
      wire#w1
      I_Contact( #LE.H )
      I_Contact( #AHLS )
      I_Contact( #Leak )
      S_Coil( #Pump_Start_A )
   END_RUNG
   RUNG wire#w1
      { S7_Templates := "SrcType := Int" } EQ_Contact(in1 := #Pump_Status, in2 := 1)
      Add(in1 := #"Step", in2 := 1, out => #"Step")
   END_RUNG
   // the same network as SCL:
   #_w1 := #"Step" = 1;
   IF #_w1 AND NOT #LE.H AND NOT #AHLS AND NOT #Leak THEN #Pump_Start_A := TRUE; END_IF;
   IF #_w1 AND (#Pump_Status = 1) THEN #"Step" := #"Step" + 1; END_IF;
END_REGION

REGION Network 3: Запуск электролизера и работа насоса
   RUNG wire#powerrail
      { S7_Templates := "SrcType := Int" } EQ_Contact(in1 := #"Step", in2 := 2)
      wire#w1
      Coil( #T_ELZ_Start.Start )
      Contact( #T_ELZ_Start."Exit" )
      I_Contact( #AHLS )
      I_Contact( #KC_1 )
      I_Contact( #KC_2 )
      I_Contact( #LE.H )
      I_Contact( #Leak )
      S_Coil( #ELZ_Start_A )
   END_RUNG
   RUNG wire#w1
      I_Contact( #AHLS )
      I_Contact( #Leak )
      S_Coil( #Pump_Start_A )
   END_RUNG
   RUNG wire#w1
      Contact( #AHLS )
      wire#w2
      R_Coil( #Pump_Start_A )
   END_RUNG
   RUNG wire#w1
      Contact( #Leak )
   END_RUNG wire#w2
   RUNG wire#w1
      I_Contact( #Start_ELZ )
      Add(in1 := #"Step", in2 := 1, out => #"Step")
   END_RUNG
   RUNG wire#w1
      Contact( #Mode )
      wire#w3
      Contact( #Gas_Chanel_1_1 )
      wire#w4
      Coil( #T_Gas.Start )
      Contact( #T_Gas."Exit" )
      S_Coil( #Gas_Stop )
      Add(in1 := #"Step", in2 := 1, out => #"Step")
   END_RUNG
   RUNG wire#w3
      Contact( #Gas_Chanel_2_1 )
   END_RUNG wire#w4
   // the same network as SCL:
   #T_ELZ_Start.Start := #"Step" = 2;
   IF #T_ELZ_Start.Start AND #T_ELZ_Start."Exit" AND NOT #AHLS AND NOT #KC_1 AND NOT #KC_2 AND NOT #LE.H AND NOT #Leak THEN
       #ELZ_Start_A := TRUE;
   END_IF;
   IF #T_ELZ_Start.Start AND NOT #AHLS AND NOT #Leak THEN #Pump_Start_A := TRUE; END_IF;
   IF #T_ELZ_Start.Start AND (#AHLS OR #Leak) THEN #Pump_Start_A := FALSE; END_IF;
   IF #T_ELZ_Start.Start AND NOT #Start_ELZ THEN #"Step" := #"Step" + 1; END_IF;
   #T_Gas.Start := #T_ELZ_Start.Start AND #Mode AND (#Gas_Chanel_1_1 OR #Gas_Chanel_2_1);
   IF #T_Gas.Start AND #T_Gas."Exit" THEN
       #Gas_Stop := TRUE;
       #"Step" := #"Step" + 1;
   END_IF;
END_REGION

REGION Network 4: Отключение электролизера
   RUNG wire#powerrail
      { S7_Templates := "SrcType := Int" } EQ_Contact(in1 := #"Step", in2 := 3)
      wire#w1
      R_Coil( #ELZ_Start_A )
   END_RUNG
   RUNG wire#w1
      { S7_Templates := "SrcType := Int" } EQ_Contact(in1 := #ELZ_Status, in2 := 0)
      Add(in1 := #"Step", in2 := 1, out => #"Step")
   END_RUNG
   // the same network as SCL:
   #_w1 := #"Step" = 3;
   IF #_w1 THEN #ELZ_Start_A := FALSE; END_IF;
   IF #_w1 AND (#ELZ_Status = 0) THEN #"Step" := #"Step" + 1; END_IF;
END_REGION

REGION Network 5: Отключение насоса
